	{attribute 'TcIecLibraryType'}
	{attribute 'external_name' := 'F_VN_RotateImageExp2_GUID_B0454A61_6B19_D120_5A5F_16C0F36D78C5'}
	(* Rotate an image by an individual rotation angle in degrees. (expert function) *)
	FUNCTION F_VN_RotateImageExp2 : HRESULT
	VAR_INPUT
		ipSrcImage	:	ITcVnImage;	(* Source image *)
		ipDestImage	:	REFERENCE TO ITcVnImage;	(* Destination image (An appropriate image will be created if required.) *)
		fAngleDeg	:	LREAL;	(* Rotation angle in degree (positive: counter-clockwise, negative: clockwise) *)
		bAdjustDestSize	:	BOOL;	(* If true, ipDestImage size is adjusted so that the whole rotated ipSrcImage is contained. Otherwise, ipDestImage size is set to ipSrcImage size. *)
		eInterpolationType	:	ETcVnInterpolationType;	(* Interpolation method *)
		eBorderInterpolation	:	ETcVnBorderInterpolationMethod;	(* Border interpolation method (ISOLATED not supported) *)
	END_VAR
	VAR_IN_OUT
		aBorderValue	:	TcVnVector4_LREAL;	(* Border value, if CONSTANT is used *)
	END_VAR
	VAR_INPUT
		hrPrev	:	HRESULT;	(* HRESULT indicating the result of previous operations (If SUCCEEDED(hrPrev) equals false, no operation is executed.) *)
	END_VAR

END_FUNCTION

// Functions/Geometric and Coordinate Transformations/F_VN_WarpAffineExp

	{attribute 'TcIecLibraryType'}
	{attribute 'external_name' := 'F_VN_WarpAffineExp_GUID_D07947C7_D823_D73C_7173_E2BD358E148A'}
	(* Apply an affine transformation to an image. (expert function) *)
	FUNCTION F_VN_WarpAffineExp : HRESULT
	VAR_INPUT
		ipSrcImage	:	ITcVnImage;	(* Source image *)
		ipDestImage	:	REFERENCE TO ITcVnImage;	(* Destination image (An appropriate image will be created if required.) *)
	END_VAR
	VAR_IN_OUT
		aTransformationMatrix	:	TcVnMatrix2x3_LREAL;	(* Affine transformation matrix *)
	END_VAR
	VAR_INPUT
		nDestWidth	:	UDINT;	(* Width of the destination image *)
		nDestHeight	:	UDINT;	(* Height of the destination image *)
		eInterpolationType	:	ETcVnInterpolationType;	(* Interpolation method *)
		bWarpInverse	:	BOOL;	(* Handle aTransformationMatrix as the inverse transformation *)
		eBorderInterpolation	:	ETcVnBorderInterpolationMethod;	(* Border interpolation method (ISOLATED not supported) *)
		fBorderValue	:	LREAL;	(* Border value, if CONSTANT is used *)
		hrPrev	:	HRESULT;	(* HRESULT indicating the result of previous operations (If SUCCEEDED(hrPrev) equals false, no operation is executed.) *)
	END_VAR

END_FUNCTION

// Functions/Geometric and Coordinate Transformations/F_VN_WarpAffine_Container

	{attribute 'TcIecLibraryType'}
	{attribute 'external_name' := 'F_VN_WarpAffine_Container_GUID_881050F9_A354_D581_448F_6DB1E8279285'}
	(* Apply an affine transformation to a container of 2D points. *)
	FUNCTION F_VN_WarpAffine_Container : HRESULT
	VAR_INPUT
		ipSrcPoints	:	ITcVnContainer;	(* Source points (ContainerType_Vector_TcVnPoint2_DINT or ContainerType_Vector_TcVnPoint2_REAL or ContainerType_Vector_TcVnPoint2_LREAL) *)
		ipDestPoints	:	REFERENCE TO ITcVnContainer;	(* Returns the transformed points (same type ID as ipSrcPoints; Non-zero interface pointers are reused.) *)
	END_VAR
	VAR_IN_OUT
		aTransformationMatrix	:	TcVnMatrix2x3_LREAL;	(* Affine transformation matrix *)
	END_VAR
	VAR_INPUT
		hrPrev	:	HRESULT;	(* HRESULT indicating the result of previous operations (If SUCCEEDED(hrPrev) equals false, no operation is executed.) *)
	END_VAR

END_FUNCTION

// Functions/Geometric and Coordinate Transformations/F_VN_WarpAffine_Point

	{attribute 'TcIecLibraryType'}
	{attribute 'external_name' := 'F_VN_WarpAffine_Point_GUID_39D72FD9_9F4F_D0F9_78FA_ACBA6F4D42D7'}
	(* Apply an affine transformation to a 2D point. *)
	FUNCTION F_VN_WarpAffine_Point : HRESULT
	VAR_IN_OUT
		aSrcPoint	:	TcVnPoint2_LREAL;	(* Source point *)
		aDestPoint	:	TcVnPoint2_LREAL;	(* Destination point *)
		aTransformationMatrix	:	TcVnMatrix2x3_LREAL;	(* Affine transformation matrix *)
	END_VAR
	VAR_INPUT
		hrPrev	:	HRESULT;	(* HRESULT indicating the result of previous operations (If SUCCEEDED(hrPrev) equals false, no operation is executed.) *)
	END_VAR

END_FUNCTION

// Functions/Geometric and Coordinate Transformations/F_VN_WarpAffine_Rectangle

	{attribute 'TcIecLibraryType'}
	{attribute 'external_name' := 'F_VN_WarpAffine_Rectangle_GUID_69BFAD85_D204_D38A_7FE5_815117E8BF2E'}
	(* Use an affine transform to warp a rectangle. *)
	FUNCTION F_VN_WarpAffine_Rectangle : HRESULT
	VAR_INPUT
		nTopLeftX	:	UDINT;	(* x coordinate of the top left corner *)
		nTopLeftY	:	UDINT;	(* y coordinate of the top left corner *)
		nBottomRightX	:	UDINT;	(* x coordinate of the bottom right corner *)
		nBottomRightY	:	UDINT;	(* y coordinate of the bottom right corner *)
		ipDestPoints	:	REFERENCE TO ITcVnContainer;	(* Returns the 4 transformed points (ContainerType_Vector_TcVnPoint2_REAL) *)
	END_VAR
	VAR_IN_OUT
		aTransformationMatrix	:	TcVnMatrix2x3_LREAL;	(* Affine transformation matrix *)
	END_VAR
	VAR_INPUT
		hrPrev	:	HRESULT;	(* HRESULT indicating the result of previous operations (If SUCCEEDED(hrPrev) equals false, no operation is executed.) *)
	END_VAR

END_FUNCTION

// Functions/Geometric and Coordinate Transformations/F_VN_WarpPerspective

	{attribute 'TcIecLibraryType'}
	{attribute 'external_name' := 'F_VN_WarpPerspective_GUID_CFE51378_A88C_D6F6_6881_5B5CC92D6876'}
	(* Apply a perspective transformation to an image. *)
	FUNCTION F_VN_WarpPerspective : HRESULT
	VAR_INPUT
		ipSrcImage	:	ITcVnImage;	(* Source image *)
		ipDestImage	:	REFERENCE TO ITcVnImage;	(* Destination image (An appropriate image will be created if required.) *)
	END_VAR
	VAR_IN_OUT
		aTransformationMatrix	:	TcVnMatrix3x3_LREAL;	(* Perspective transformation matrix *)
	END_VAR
	VAR_INPUT
		hrPrev	:	HRESULT;	(* HRESULT indicating the result of previous operations (If SUCCEEDED(hrPrev) equals false, no operation is executed.) *)
	END_VAR

END_FUNCTION

// Functions/Geometric and Coordinate Transformations/F_VN_WarpPerspective_Container

	{attribute 'TcIecLibraryType'}
	{attribute 'external_name' := 'F_VN_WarpPerspective_Container_GUID_C43078FC_8F1A_D906_4EBD_0A8B2D834094'}
	(* Apply a perspective transformation to a container of 2D points. *)
	FUNCTION F_VN_WarpPerspective_Container : HRESULT
	VAR_INPUT
		ipSrcPoints	:	ITcVnContainer;	(* Source points (ContainerType_Vector_TcVnPoint2_DINT or ContainerType_Vector_TcVnPoint2_REAL or ContainerType_Vector_TcVnPoint2_LREAL) *)
		ipDestPoints	:	REFERENCE TO ITcVnContainer;	(* Returns the transformed points (same type ID as ipSrcPoints; Non-zero interface pointers are reused.) *)
	END_VAR
	VAR_IN_OUT
		aTransformationMatrix	:	TcVnMatrix3x3_LREAL;	(* Perspective transformation matrix *)
	END_VAR
	VAR_INPUT
		hrPrev	:	HRESULT;	(* HRESULT indicating the result of previous operations (If SUCCEEDED(hrPrev) equals false, no operation is executed.) *)
	END_VAR

END_FUNCTION

// Functions/Geometric and Coordinate Transformations/F_VN_WarpPerspectiveExp

	{attribute 'TcIecLibraryType'}
	{attribute 'external_name' := 'F_VN_WarpPerspectiveExp_GUID_34B331D2_78AA_D3E3_7DC8_94B3A3627598'}
	(* Apply a perspective transformation to an image. (expert function) *)
	FUNCTION F_VN_WarpPerspectiveExp : HRESULT
	VAR_INPUT
		ipSrcImage	:	ITcVnImage;	(* Source image *)
		ipDestImage	:	REFERENCE TO ITcVnImage;	(* Destination image (An appropriate image will be created if required.) *)
	END_VAR
	VAR_IN_OUT
		aTransformationMatrix	:	TcVnMatrix3x3_LREAL;	(* Perspective transformation matrix *)
	END_VAR
	VAR_INPUT
		nDestWidth	:	UDINT;	(* Width of the destination image *)
		nDestHeight	:	UDINT;	(* Height of the destination image *)
		eInterpolationType	:	ETcVnInterpolationType;	(* Interpolation method *)
		bWarpInverse	:	BOOL;	(* Handle aTransformationMatrix as the inverse transformation *)
		eBorderInterpolation	:	ETcVnBorderInterpolationMethod;	(* Border interpolation method (ISOLATED not supported) *)
		fBorderValue	:	LREAL;	(* Border value, if CONSTANT is used *)
		hrPrev	:	HRESULT;	(* HRESULT indicating the result of previous operations (If SUCCEEDED(hrPrev) equals false, no operation is executed.) *)
	END_VAR

END_FUNCTION

// Functions/Geometric and Coordinate Transformations/F_VN_WarpPerspective_Point

	{attribute 'TcIecLibraryType'}
	{attribute 'external_name' := 'F_VN_WarpPerspective_Point_GUID_3F6D0E94_50F7_D140_62FB_6E3EA1ADD95E'}
	(* Apply a perspective transformation to a 2D point. *)
	FUNCTION F_VN_WarpPerspective_Point : HRESULT
	VAR_IN_OUT
		aSrcPoint	:	TcVnPoint2_LREAL;	(* Source point *)
		aDestPoint	:	TcVnPoint2_LREAL;	(* Destination point *)
		aTransformationMatrix	:	TcVnMatrix3x3_LREAL;	(* Perspective transformation matrix *)
	END_VAR
	VAR_INPUT
		hrPrev	:	HRESULT;	(* HRESULT indicating the result of previous operations (If SUCCEEDED(hrPrev) equals false, no operation is executed.) *)
	END_VAR

END_FUNCTION

// Functions/Geometric and Coordinate Transformations/F_VN_WarpPerspective_Rectangle

	{attribute 'TcIecLibraryType'}
	{attribute 'external_name' := 'F_VN_WarpPerspective_Rectangle_GUID_C900301F_B0CF_D57A_7958_23BC0F26B8F7'}
	(* Use a perspective transform to warp a rectangle. *)
	FUNCTION F_VN_WarpPerspective_Rectangle : HRESULT
	VAR_INPUT
		nTopLeftX	:	UDINT;	(* x coordinate of the top left corner *)
		nTopLeftY	:	UDINT;	(* y coordinate of the top left corner *)
		nBottomRightX	:	UDINT;	(* x coordinate of the bottom right corner *)
		nBottomRightY	:	UDINT;	(* y coordinate of the bottom right corner *)
		ipDestPoints	:	REFERENCE TO ITcVnContainer;	(* Returns the 4 transformed points (ContainerType_Vector_TcVnPoint2_REAL) *)
	END_VAR
	VAR_IN_OUT
		aTransformationMatrix	:	TcVnMatrix3x3_LREAL;	(* Perspective transformation matrix *)
	END_VAR
	VAR_INPUT
		hrPrev	:	HRESULT;	(* HRESULT indicating the result of previous operations (If SUCCEEDED(hrPrev) equals false, no operation is executed.) *)
	END_VAR

END_FUNCTION

// Functions/Image Color and Contrast Processing/F_VN_ApplyColorMap

	{attribute 'TcIecLibraryType'}
	{attribute 'external_name' := 'F_VN_ApplyColorMap_GUID_5FC1F56C_5B3C_D465_60AA_C4AA3854379F'}
	(* Apply a color map to a gray-level image. *)
	FUNCTION F_VN_ApplyColorMap : HRESULT
	VAR_INPUT
		ipSrcImage	:	ITcVnImage;	(* Source image (TCVN_ET_USINT or TCVN_ET_UINT, 1 channel) *)
		ipDestImage	:	REFERENCE TO ITcVnImage;	(* Returns the colored image (TCVN_ET_USINT, 3 channel. An appropriate image will be created if required.) *)
		ipColorMap	:	ITcVnContainer;	(* Color map to be applied to ipSrcImage (ContainerType_Vector_TcVnVector3_REAL with 256 or 65536 elements, dependent on ipSrcImage type). Can be either custom or created with F_VN_GenerateColorMap. *)
		hrPrev	:	HRESULT;	(* HRESULT indicating the result of previous operations (If SUCCEEDED(hrPrev) equals false, no operation is executed.) *)
	END_VAR

END_FUNCTION

// Functions/Image Color and Contrast Processing/F_VN_GenerateColorMap

	{attribute 'TcIecLibraryType'}
	{attribute 'external_name' := 'F_VN_GenerateColorMap_GUID_41124A2C_62FC_DD0A_4BF9_B43C26A42D18'}
	(* Generates a pre-defined color map. *)
	FUNCTION F_VN_GenerateColorMap : HRESULT
	VAR_INPUT
		ipColorMap	:	REFERENCE TO ITcVnContainer;	(* Returns the color map (ContainerType_Vector_TcVnVector3_REAL with 256 or 65536 elements) *)
		eColorMap	:	ETcVnColorMap;	(* Selects a color map (similar to GNU Octave/MATLAB types) *)
		eColorMapSize	:	ETcVnColorMapSize;	(* Defines how many elements the generated color map should have *)
		hrPrev	:	HRESULT;	(* HRESULT indicating the result of previous operations (If SUCCEEDED(hrPrev) equals false, no operation is executed.) *)
	END_VAR

END_FUNCTION

// Functions/Image Color and Contrast Processing/F_VN_ApplyLut

	{attribute 'TcIecLibraryType'}
	{attribute 'external_name' := 'F_VN_ApplyLut_GUID_5D73781A_C824_D04E_6F7A_A9EAA2AB4681'}
	(* Apply a lookup table to an image to manipulate its colors. *)
	FUNCTION F_VN_ApplyLut : HRESULT
	VAR_INPUT
		ipSrcImage	:	ITcVnImage;	(* Source image (1-4 channels of 8 or 16 bit types SINT, USINT, INT, UINT) *)
		ipDestImage	:	REFERENCE TO ITcVnImage;	(* Returns the result image (same size, type and channels as ipSrcImage. An appropriate image will be created if required.) *)
		ipLut	:	ITcVnContainer;	(* Lookup table with elements matching ipSrcImage type and either 256 (8 bit images) or 65536 (16 bit images) elements. E.g. ContainerType_Vector_USINT for 1-4 channel USINT image (in this case, the same lookup values are used for each channel) or ContainerType_Vector_TcVnVector3_USINT for a 3 channel USINT image (in this case, each channel uses an individual lookup value).
						 *)
		hrPrev	:	HRESULT;	(* HRESULT indicating the result of previous operations (If SUCCEEDED(hrPrev) equals false, no operation is executed.) *)
	END_VAR

END_FUNCTION

// Functions/Image Color and Contrast Processing/F_VN_Clahe

	{attribute 'TcIecLibraryType'}
	{attribute 'external_name' := 'F_VN_Clahe_GUID_6F92982A_1259_D9E8_5872_BC9EEE361F4F'}
	(* Apply Constrast Limited Adaptive Histogram Equalization. This applies local histogram equalization to individual tiles. *)
	FUNCTION F_VN_Clahe : HRESULT
	VAR_INPUT
		ipSrcImage	:	ITcVnImage;	(* Source image (TCVN_ET_USINT or TCVN_ET_UINT, 1 channel) *)
		ipDestImage	:	REFERENCE TO ITcVnImage;	(* Returns the resulting image (An appropriate image will be created if required.) *)
		hrPrev	:	HRESULT;	(* HRESULT indicating the result of previous operations (If SUCCEEDED(hrPrev) equals false, no operation is executed.) *)
	END_VAR

END_FUNCTION

// Functions/Image Color and Contrast Processing/F_VN_ClaheExp

	{attribute 'TcIecLibraryType'}
	{attribute 'external_name' := 'F_VN_ClaheExp_GUID_D5AEAD88_7973_D98E_640E_FCB90EEA4C61'}
	(* Apply Constrast Limited Adaptive Histogram Equalization. This applies local histogram equalization to individual tiles. (expert function) *)
	FUNCTION F_VN_ClaheExp : HRESULT
	VAR_INPUT
		ipSrcImage	:	ITcVnImage;	(* Source image (TCVN_ET_USINT or TCVN_ET_UINT, 1 channel) *)
		ipDestImage	:	REFERENCE TO ITcVnImage;	(* Returns the resulting image (An appropriate image will be created if required.) *)
		fClipLimit	:	LREAL;	(* Threshold for contrast limit (set to <= 0 to disable clipping) *)
		nTilesX	:	UDINT;	(* Number of tiles in x direction *)
		nTilesY	:	UDINT;	(* Number of tiles in y direction *)
		hrPrev	:	HRESULT;	(* HRESULT indicating the result of previous operations (If SUCCEEDED(hrPrev) equals false, no operation is executed.) *)
	END_VAR

END_FUNCTION

// Functions/Image Color and Contrast Processing/F_VN_ConvertColorSpace

	{attribute 'TcIecLibraryType'}
	{attribute 'external_name' := 'F_VN_ConvertColorSpace_GUID_3928ED09_5286_D091_6CFF_018E8A67A19B'}
	(* Convert image from one color space to another. *)
	FUNCTION F_VN_ConvertColorSpace : HRESULT
	VAR_INPUT
		ipSrcImage	:	ITcVnImage;	(* Source image *)
		ipDestImage	:	REFERENCE TO ITcVnImage;	(* Destination image (An appropriate destination image will be created if required.) *)
		eTransform	:	ETcVnColorSpaceTransform;	(* Transforms to be applied *)
		hrPrev	:	HRESULT;	(* HRESULT indicating the result of previous operations (If SUCCEEDED(hrPrev) equals false, no operation is executed.) *)
	END_VAR

END_FUNCTION

// Functions/Image Color and Contrast Processing/F_VN_GenerateCustomColorMap

	{attribute 'TcIecLibraryType'}
	{attribute 'external_name' := 'F_VN_GenerateCustomColorMap_GUID_25265482_D991_DD20_5A65_7D8187FF081F'}
	(* Generate a custom color map by interpolating between user defined colors (equally distributed, linear for each channel). *)
	FUNCTION F_VN_GenerateCustomColorMap : HRESULT
	VAR_INPUT
		ipColorMap	:	REFERENCE TO ITcVnContainer;	(* Returns the color map (ContainerType_Vector_TcVnVector3_REAL with 256 or 65536 elements) *)
		ipInitialColors	:	ITcVnContainer;	(* User defined colors (ContainerType_Vector_TcVnVector3_REAL, at least 2 elements) *)
		eColorMapSize	:	ETcVnColorMapSize;	(* Defines how many elements the generated color map should have *)
		hrPrev	:	HRESULT;	(* HRESULT indicating the result of previous operations (If SUCCEEDED(hrPrev) equals false, no operation is executed.) *)
	END_VAR

END_FUNCTION

// Functions/Image Color and Contrast Processing/F_VN_Histogram

	{attribute 'TcIecLibraryType'}
	{attribute 'external_name' := 'F_VN_Histogram_GUID_4967AB6E_7C40_DDEE_7ACD_6DC0B6B84EBF'}
	(* Calculate the (multi-channel) histogram of an image. *)
	FUNCTION F_VN_Histogram : HRESULT
	VAR_INPUT
		ipSrcImage	:	ITcVnImage;	(* Source image *)
		ipDestHistogram	:	REFERENCE TO ITcVnContainer;	(* Returns a container with a multi-channel histogram, where every channel is represented as a vector of UDINT (ContainerType_Vector_Vector_UDINT. Non-zero interface pointers are reused.) *)
		hrPrev	:	HRESULT;	(* HRESULT indicating the result of previous operations (If SUCCEEDED(hrPrev) equals false, no operation is executed.) *)
	END_VAR

END_FUNCTION

// Functions/Image Color and Contrast Processing/F_VN_HistogramExp

	{attribute 'TcIecLibraryType'}
	{attribute 'external_name' := 'F_VN_HistogramExp_GUID_C24DCAD7_922F_DA99_5C1A_00E5A61DD4E7'}
	(* Calculate the (multi-channel) histogram of an image. (expert function) *)
	FUNCTION F_VN_HistogramExp : HRESULT
	VAR_INPUT
		ipSrcImage	:	ITcVnImage;	(* Source image *)
		ipDestHistogram	:	REFERENCE TO ITcVnContainer;	(* Returns a container with a multi-channel histogram, where every channel is represented as a vector of UDINT (ContainerType_Vector_Vector_UDINT. Non-zero interface pointers are reused.) *)
	END_VAR
	VAR_IN_OUT
		nBins	:	UDINT;	(* Desired number of bins or 0 to keep the default for the corresponding image format (in) and default number of bins (out) *)
		fLowerBound	:	LREAL;	(* Lower (inclusive) boundary of the 0-th histogram bin (in), or receive the default if fLowerBound AND fUpperBound are set to 0 (out) *)
		fUpperBound	:	LREAL;	(* Upper (exclusive) boundary of the last histogram bin nBins-1 (in), or receive the default if fLowerBound AND fUpperBound are set to 0 (out) *)
	END_VAR
	VAR_INPUT
		ipMask	:	ITcVnImage;	(* Source image mask (TCVN_ET_USINT, 1 channel. Mask is optional, set to 0 if not required.) *)
		hrPrev	:	HRESULT;	(* HRESULT indicating the result of previous operations (If SUCCEEDED(hrPrev) equals false, no operation is executed.) *)
	END_VAR

END_FUNCTION

// Functions/Image Color and Contrast Processing/F_VN_HistogramEqualization

	{attribute 'TcIecLibraryType'}
	{attribute 'external_name' := 'F_VN_HistogramEqualization_GUID_E4A7191D_DEB2_D844_61A1_8D5192620F8A'}
	(* Equalize the histogram of a grayscale or rgb image, which normalizes the brightness and improves the contrast. *)
	FUNCTION F_VN_HistogramEqualization : HRESULT
	VAR_INPUT
		ipSrcImage	:	ITcVnImage;	(* Source image *)
		ipDestImage	:	REFERENCE TO ITcVnImage;	(* Destination image (An appropriate destination image will be created if required.) *)
		hrPrev	:	HRESULT;	(* HRESULT indicating the result of previous operations (If SUCCEEDED(hrPrev) equals false, no operation is executed.) *)
	END_VAR

END_FUNCTION

// Functions/Image Color and Contrast Processing/F_VN_HistogramEqualizationExp

	{attribute 'TcIecLibraryType'}
	{attribute 'external_name' := 'F_VN_HistogramEqualizationExp_GUID_8EB4C057_2479_D74C_4CCA_F2B7F514C2BC'}
	(* Equalize the histogram of a grayscale or color image, which normalizes the brightness and improves the contrast. (expert function) 
	The channel index that should be equalized has to be specified (-1 expects a RGB image, converts it to YCbCr, equalizes the Y channel and converts the image back to RGB).  *)
	FUNCTION F_VN_HistogramEqualizationExp : HRESULT
	VAR_INPUT
		ipSrcImage	:	ITcVnImage;	(* Source image *)
		ipDestImage	:	REFERENCE TO ITcVnImage;	(* Destination image (An appropriate destination image will be created if required.) *)
		nChannelIdx	:	INT;	(* Index of the image channel that should be equalized (-1 expects a RGB image, converts it to YCbCr, equalizes the Y channel and converts the image back to RGB) *)
		hrPrev	:	HRESULT;	(* HRESULT indicating the result of previous operations (If SUCCEEDED(hrPrev) equals false, no operation is executed.) *)
	END_VAR

END_FUNCTION

// Functions/Image Color and Contrast Processing/F_VN_InvertImageColor

	{attribute 'TcIecLibraryType'}
	{attribute 'external_name' := 'F_VN_InvertImageColor_GUID_37BC3565_41C2_D780_6FEB_8C8E78361D97'}
	(* Invert the color of an image.
          For signed integer or negative floating point values, only the signs will be switched.
          If the image contains only positive floating point values, each pixel value is subtracted from the maximum available pixel value (or 1.0, whatever is higher). *)
	FUNCTION F_VN_InvertImageColor : HRESULT
	VAR_INPUT
		ipSrcImage	:	ITcVnImage;	(* Source image *)
		ipDestImage	:	REFERENCE TO ITcVnImage;	(* Destination image (An appropriate image will be created if required.) *)
		hrPrev	:	HRESULT;	(* HRESULT indicating the result of previous operations (If SUCCEEDED(hrPrev) equals false, no operation is executed.) *)
	END_VAR

END_FUNCTION

// Functions/Image Color and Contrast Processing/F_VN_InvertImageColorExp

	{attribute 'TcIecLibraryType'}
	{attribute 'external_name' := 'F_VN_InvertImageColorExp_GUID_D8CA267F_20FA_D72A_5CA4_D061DDB2DC5B'}
	(* Invert the color of an image. (expert function)
          For signed integer or negative floating point values, only the signs will be switched.
          If the image contains only positive floating point values, each pixel value is subtracted from the maximum available pixel value (or 1.0, whatever is higher). *)
	FUNCTION F_VN_InvertImageColorExp : HRESULT
	VAR_INPUT
		ipSrcImage	:	ITcVnImage;	(* Source image *)
		ipDestImage	:	REFERENCE TO ITcVnImage;	(* Destination image (An appropriate image will be created if required.) *)
		fMaxValue	:	LREAL;	(* Maximum pixel value (e.g. if a 16 bit image contains 12 bit values). -1 means the default values are used. *)
		hrPrev	:	HRESULT;	(* HRESULT indicating the result of previous operations (If SUCCEEDED(hrPrev) equals false, no operation is executed.) *)
	END_VAR

END_FUNCTION

// Functions/Image Color and Contrast Processing/F_VN_NormalizeImage

	{attribute 'TcIecLibraryType'}
	{attribute 'external_name' := 'F_VN_NormalizeImage_GUID_01C94C10_A06A_D62A_55A0_B2526D33140F'}
	(* Normalize an image regarding its value range (e.g. stretch pixel values [50..150] to full range [0..255]). *)
	FUNCTION F_VN_NormalizeImage : HRESULT
	VAR_INPUT
		ipSrcImage	:	ITcVnImage;	(* Source image *)
		ipDestImage	:	REFERENCE TO ITcVnImage;	(* Destination image (An appropriate destination image will be created if required.) *)
		hrPrev	:	HRESULT;	(* HRESULT indicating the result of previous operations (If SUCCEEDED(hrPrev) equals false, no operation is executed.) *)
	END_VAR

END_FUNCTION

// Functions/Image Color and Contrast Processing/F_VN_NormalizeImageExp

	{attribute 'TcIecLibraryType'}
	{attribute 'external_name' := 'F_VN_NormalizeImageExp_GUID_F9250BFC_E526_D3A0_70B1_145F0908CE43'}
	(* Normalize an image regarding its value range (e.g. stretch pixel values [50..150] to full range [0..255]) or scale the values regarding a specific normalization (e.g. L2-norm). (expert function) *)
	FUNCTION F_VN_NormalizeImageExp : HRESULT
	VAR_INPUT
		ipSrcImage	:	ITcVnImage;	(* Source image *)
		ipDestImage	:	REFERENCE TO ITcVnImage;	(* Destination image (An appropriate destination image will be created if required.) *)
		fAlpha	:	LREAL;	(* Lower range boundary (in case of normalizing the value range) or value to normalize to (||ipDestImage|| = fAlpha) *)
		fBeta	:	LREAL;	(* Upper range boundary (in case of normalizing the value range) *)
		eNormType	:	ETcVnNormalizationType;	(* Normalization type (only INF, L1, L2 or MINMAX) *)
		eDestType	:	ETcVnElementType;	(* Destination image depth (usually SAME_AS_SOURCE) *)
		ipMask	:	ITcVnImage;	(* Mask to restrict the normalization to specific pixel positions (set 0 to normalize the whole image) *)
		hrPrev	:	HRESULT;	(* HRESULT indicating the result of previous operations (If SUCCEEDED(hrPrev) equals false, no operation is executed.) *)
	END_VAR

END_FUNCTION

// Functions/Image Color and Contrast Processing/F_VN_NormalizeImageForDisplay

	{attribute 'TcIecLibraryType'}
	{attribute 'external_name' := 'F_VN_NormalizeImageForDisplay_GUID_5A39AF93_6FA8_DA77_5213_DA2C848DE791'}
	(* Normalize an image for display, i.e. scale it to the full value range of the underlying data type (-1 to 1 for floating point). *)
	FUNCTION F_VN_NormalizeImageForDisplay : HRESULT
	VAR_INPUT
		ipSrcImage	:	ITcVnImage;	(* Source image *)
		ipDestImage	:	REFERENCE TO ITcVnImage;	(* Destination image (An appropriate destination image will be created if required.) *)
		eSignedNormalization	:	ETcVnSignedNormalization;	(* Option for normalizing signed values *)
		hrPrev	:	HRESULT;	(* HRESULT indicating the result of previous operations (If SUCCEEDED(hrPrev) equals false, no operation is executed.) *)
	END_VAR

END_FUNCTION

// Functions/Image Color and Contrast Processing/F_VN_ReferenceColorSimilarity_ITcVnColorModel

	{attribute 'TcIecLibraryType'}
	{attribute 'external_name' := 'F_VN_ReferenceColorSimilarity_ITcVnColorModel_GUID_2A1F7AC8_C700_D330_6AC5_E4FDC13D131C'}
	(* Computes the similarity to a reference color model for each pixel in the source image. *)
	FUNCTION F_VN_ReferenceColorSimilarity_ITcVnColorModel : HRESULT
	VAR_INPUT
		ipSrcImage	:	ITcVnImage;	(* RGB source image (USINT, 3 channels) *)
		ipDestImage	:	REFERENCE TO ITcVnImage;	(* Returns the similarity to ipColorModel for each pixel in ipSrcImage (USINT, 1 channel. An appropriate destination image will be created if required.) *)
		ipColorModel	:	ITcVnColorModel;	(* Color model *)
		hrPrev	:	HRESULT;	(* HRESULT indicating the result of previous operations (If SUCCEEDED(hrPrev) equals false, no operation is executed.) *)
	END_VAR

END_FUNCTION

// Interfaces/Machine Learning/ITcVnColorModel

	(* Interface to train and classify an image color. *)
	{attribute 'c++_compatible'}
	{attribute 'vtable_order' := 'TrainImageColor;ClassifyImageColor'}
	INTERFACE ITcVnColorModel EXTENDS ITcVnMlModel


(* Train the color of the provided image. *)
	{attribute 'c++_compatible'}
	{attribute 'minimal_input_size' := '4'}
	{attribute 'pack_mode' := '4'}
	METHOD TrainImageColor : HRESULT
	VAR_INPUT
		ipSrcImage : ITcVnImage;
		nDifferentColors : UDINT;
		ipMask : ITcVnImage;
		nSkipPixels : UDINT;
	END_VAR
END_METHOD


(* Compute the similarity of each image pixel to the trained reference color. *)
	{attribute 'c++_compatible'}
	{attribute 'minimal_input_size' := '4'}
	{attribute 'pack_mode' := '4'}
	METHOD ClassifyImageColor : HRESULT
	VAR_INPUT
		ipSrcImage : ITcVnImage;
		pipDestImage : POINTER TO ITcVnImage;
		fVariance : REAL;
		fLuminanceWeight : REAL;
	END_VAR
END_METHOD

END_INTERFACE

// Functions/Image Color and Contrast Processing/F_VN_ReferenceColorSimilarityExp_ITcVnColorModel

	{attribute 'TcIecLibraryType'}
	{attribute 'external_name' := 'F_VN_ReferenceColorSimilarityExp_ITcVnColorModel_GUID_2E034A73_4EF1_D287_407C_3A587C275268'}
	(* Computes the similarity to a reference color model for each pixel in the source image. (expert function) *)
	FUNCTION F_VN_ReferenceColorSimilarityExp_ITcVnColorModel : HRESULT
	VAR_INPUT
		ipSrcImage	:	ITcVnImage;	(* RGB source image (USINT, 3 channels) *)
		ipDestImage	:	REFERENCE TO ITcVnImage;	(* Returns the similarity to ipColorModel for each pixel in ipSrcImage (USINT, 1 channel. An appropriate destination image will be created if required.) *)
		ipColorModel	:	ITcVnColorModel;	(* Color model *)
		fVariance	:	REAL;	(* Allowed color variance (0.1 - 0.3 might be a good start to try) *)
		fLuminanceWeight	:	REAL;	(* Weight the impact of the luminance ([0..1], e.g. set to 0 to be more resistant to unequal illumination, but might be required to differentiate between some colors. Ignored if ipColorModel is of type RGB.) *)
		hrPrev	:	HRESULT;	(* HRESULT indicating the result of previous operations (If SUCCEEDED(hrPrev) equals false, no operation is executed.) *)
	END_VAR

END_FUNCTION

// Functions/Image Color and Contrast Processing/F_VN_ReferenceColorSimilarity_ITcVnMlModel

	{attribute 'TcIecLibraryType'}
	{attribute 'external_name' := 'F_VN_ReferenceColorSimilarity_ITcVnMlModel_GUID_7A720166_859C_DC02_5DA3_02CED4582008'}
	(* Computes the similarity to a reference color model for each pixel in the source image. *)
	FUNCTION F_VN_ReferenceColorSimilarity_ITcVnMlModel : HRESULT
	VAR_INPUT
		ipSrcImage	:	ITcVnImage;	(* RGB source image (USINT, 3 channels) *)
		ipDestImage	:	REFERENCE TO ITcVnImage;	(* Returns the similarity to ipColorModel for each pixel in ipSrcImage (USINT, 1 channel. An appropriate destination image will be created if required.) *)
		ipColorModel	:	ITcVnMlModel;	(* Color model *)
		hrPrev	:	HRESULT;	(* HRESULT indicating the result of previous operations (If SUCCEEDED(hrPrev) equals false, no operation is executed.) *)
	END_VAR

END_FUNCTION

// Functions/Image Color and Contrast Processing/F_VN_ReferenceColorSimilarityExp_ITcVnMlModel

	{attribute 'TcIecLibraryType'}
	{attribute 'external_name' := 'F_VN_ReferenceColorSimilarityExp_ITcVnMlModel_GUID_58AE79C4_8392_D997_6DCA_D06724B6AE4D'}
	(* Computes the similarity to a reference color model for each pixel in the source image. (expert function) *)
	FUNCTION F_VN_ReferenceColorSimilarityExp_ITcVnMlModel : HRESULT
	VAR_INPUT
		ipSrcImage	:	ITcVnImage;	(* RGB source image (USINT, 3 channels) *)
		ipDestImage	:	REFERENCE TO ITcVnImage;	(* Returns the similarity to ipColorModel for each pixel in ipSrcImage (USINT, 1 channel. An appropriate destination image will be created if required.) *)
		ipColorModel	:	ITcVnMlModel;	(* Color model *)
		fVariance	:	REAL;	(* Allowed color variance (0.1 - 0.3 might be a good start to try) *)
		fLuminanceWeight	:	REAL;	(* Weight the impact of the luminance ([0..1], e.g. set to 0 to be more resistant to unequal illumination, but might be required to differentiate between some colors. Ignored if ipColorModel is of type RGB.) *)
		hrPrev	:	HRESULT;	(* HRESULT indicating the result of previous operations (If SUCCEEDED(hrPrev) equals false, no operation is executed.) *)
	END_VAR

END_FUNCTION

// Functions/Image Color and Contrast Processing/F_VN_ReferenceColorSimilarity_TcVnVector3_LREAL

	{attribute 'TcIecLibraryType'}
	{attribute 'external_name' := 'F_VN_ReferenceColorSimilarity_TcVnVector3_LREAL_GUID_FAFF8BBB_F60C_DAC4_5500_10EB08A58633'}
	(* Computes the similarity to a reference color for each pixel in the source image. *)
	FUNCTION F_VN_ReferenceColorSimilarity_TcVnVector3_LREAL : HRESULT
	VAR_INPUT
		ipSrcImage	:	ITcVnImage;	(* RGB source image (USINT, 3 channels) *)
		ipDestImage	:	REFERENCE TO ITcVnImage;	(* Returns the similarity to aRefColor for each pixel in ipSrcImage (USINT, 1 channel. An appropriate destination image will be created if required.) *)
	END_VAR
	VAR_IN_OUT
		aRefColor	:	TcVnVector3_LREAL;	(* Reference color (RGB, [0..255]) *)
	END_VAR
	VAR_INPUT
		hrPrev	:	HRESULT;	(* HRESULT indicating the result of previous operations (If SUCCEEDED(hrPrev) equals false, no operation is executed.) *)
	END_VAR

END_FUNCTION

// Functions/Image Color and Contrast Processing/F_VN_ReferenceColorSimilarityExp_TcVnVector3_LREAL

	{attribute 'TcIecLibraryType'}
	{attribute 'external_name' := 'F_VN_ReferenceColorSimilarityExp_TcVnVector3_LREAL_GUID_D374A0BE_D5EA_D011_61D8_43F8E1C41E27'}
	(* Computes the similarity to a reference color for each pixel in the source image. (expert function) *)
	FUNCTION F_VN_ReferenceColorSimilarityExp_TcVnVector3_LREAL : HRESULT
	VAR_INPUT
		ipSrcImage	:	ITcVnImage;	(* RGB source image (USINT, 3 channels) *)
		ipDestImage	:	REFERENCE TO ITcVnImage;	(* Returns the similarity to aRefColor for each pixel in ipSrcImage (USINT, 1 channel. An appropriate destination image will be created if required.) *)
	END_VAR
	VAR_IN_OUT
		aRefColor	:	TcVnVector3_LREAL;	(* Reference color (RGB, [0..255]) *)
	END_VAR
	VAR_INPUT
		fVariance	:	REAL;	(* Allowed color variance (0.1 - 0.3 might be a good start to try) *)
		fLuminanceWeight	:	REAL;	(* Weight the impact of the luminance ([0..1], e.g. set to 0 to be more resistant to unequal illumination, but might be required to differentiate between some colors) *)
		hrPrev	:	HRESULT;	(* HRESULT indicating the result of previous operations (If SUCCEEDED(hrPrev) equals false, no operation is executed.) *)
	END_VAR

END_FUNCTION

// Functions/Image Color and Contrast Processing/F_VN_TrainImageColor

	{attribute 'TcIecLibraryType'}
	{attribute 'external_name' := 'F_VN_TrainImageColor_GUID_0286D650_F00C_DA59_6156_CB0B6313F883'}
	(* Create a new color model, describing the image color. *)
	FUNCTION F_VN_TrainImageColor : HRESULT
	VAR_INPUT
		ipSrcImage	:	ITcVnImage;	(* Source image (3 channels (RGB) of type USINT) *)
		ipColorModel	:	REFERENCE TO ITcVnColorModel;	(* Returns the color model *)
		nDifferentColors	:	UDINT;	(* Number of different colors to distinguish *)
		hrPrev	:	HRESULT;	(* HRESULT indicating the result of previous operations (If SUCCEEDED(hrPrev) equals false, no operation is executed.) *)
	END_VAR

END_FUNCTION

// Functions/Image Color and Contrast Processing/F_VN_TrainImageColorExp

	{attribute 'TcIecLibraryType'}
	{attribute 'external_name' := 'F_VN_TrainImageColorExp_GUID_615355F9_6BAF_DD2B_4648_974DBAB6D17A'}
	(* Create a new color model, describing the image color. (expert function) *)
	FUNCTION F_VN_TrainImageColorExp : HRESULT
	VAR_INPUT
		ipSrcImage	:	ITcVnImage;	(* Source image (3 channels (RGB) of type USINT) *)
		ipColorModel	:	REFERENCE TO ITcVnColorModel;	(* Returns the color model *)
		nDifferentColors	:	UDINT;	(* Number of different colors to distinguish *)
		eMethod	:	ETcVnColorTrainingMethod;	(* Color training method *)
		ipMask	:	ITcVnImage;	(* Optional image mask (1 channel of type USINT, set to 0 if not required) *)
		nSkipPixels	:	UDINT;	(* Number of pixels to skip between each evaluated color sample (to achieve a better performance). 0 takes every pixel into account and tends to be more accurate. *)
		hrPrev	:	HRESULT;	(* HRESULT indicating the result of previous operations (If SUCCEEDED(hrPrev) equals false, no operation is executed.) *)
	END_VAR

END_FUNCTION

// Functions/Image Color and Contrast Processing/F_VN_TrainImageColorExp2

	{attribute 'TcIecLibraryType'}
	{attribute 'external_name' := 'F_VN_TrainImageColorExp2_GUID_04621000_6349_D589_543F_EA070237B42C'}
	(* Create a new color model, describing the image color. (expert function) *)
	FUNCTION F_VN_TrainImageColorExp2 : HRESULT
	VAR_INPUT
		ipSrcImage	:	ITcVnImage;	(* Source image (3 channels (RGB) of type USINT) *)
		ipColorModel	:	REFERENCE TO ITcVnColorModel;	(* Returns the color model *)
		nDifferentColors	:	UDINT;	(* Maximum number of different colors to distinguish (if LBG is used as a clustering algorithm, the result might have less different colors, depending on nMaxClusterRadius) *)
		eMethod	:	ETcVnColorTrainingMethod;	(* Color training method *)
		ipMask	:	ITcVnImage;	(* Optional image mask (1 channel of type USINT, set to 0 if not required) *)
		nSkipPixels	:	UDINT;	(* Number of pixels to skip between each evaluated color sample (to achieve a better performance). 0 takes every pixel into account and tends to be more accurate. *)
		eClusteringAlgorithm	:	ETcVnClusteringAlgorithm;	(* Clustering algorithm *)
		nMaxClusterRadius	:	DINT;	(* Only used for the LBG clustering algorithm. Maximum allowed radius (> 0) of a single cluster, i.e. clusters with a higher radius will be split into smaller ones, until a global number of nDifferentColors is reached. *)
		bSingleSplitSteps	:	BOOL;	(* Only used for the LBG clustering algorithm. If true, the global optimization is always run after a single cluster has been split. If false, several clusters are split within the same step before applying the global optimization. Applying the global optimization less often is faster, but can lead to less optimal results, especially having 2 nearby clusters that could be represented by 1) *)
		hrPrev	:	HRESULT;	(* HRESULT indicating the result of previous operations (If SUCCEEDED(hrPrev) equals false, no operation is executed.) *)
	END_VAR

END_FUNCTION

// Functions/Image Color and Contrast Processing/F_VN_TrainImageColor_ITcVnMlModel

	{attribute 'TcIecLibraryType'}
	{attribute 'external_name' := 'F_VN_TrainImageColor_ITcVnMlModel_GUID_4985D650_730F_DDD3_537C_883607504684'}
	(* Create a new color model, describing the image color. *)
	FUNCTION F_VN_TrainImageColor_ITcVnMlModel : HRESULT
	VAR_INPUT
		ipSrcImage	:	ITcVnImage;	(* Source image (3 channels (RGB) of type USINT) *)
		ipColorModel	:	REFERENCE TO ITcVnMlModel;	(* Returns the color model *)
		nDifferentColors	:	UDINT;	(* Number of different colors to distinguish *)
		hrPrev	:	HRESULT;	(* HRESULT indicating the result of previous operations (If SUCCEEDED(hrPrev) equals false, no operation is executed.) *)
	END_VAR

END_FUNCTION

// Functions/Image Color and Contrast Processing/F_VN_TrainImageColorExp_ITcVnMlModel

	{attribute 'TcIecLibraryType'}
	{attribute 'external_name' := 'F_VN_TrainImageColorExp_ITcVnMlModel_GUID_EA6BA25E_3C46_DF47_6C6F_22F5A52F9D7A'}
	(* Create a new color model, describing the image color. (expert function) *)
	FUNCTION F_VN_TrainImageColorExp_ITcVnMlModel : HRESULT
	VAR_INPUT
		ipSrcImage	:	ITcVnImage;	(* Source image (3 channels (RGB) of type USINT) *)
		ipColorModel	:	REFERENCE TO ITcVnMlModel;	(* Returns the color model *)
		nDifferentColors	:	UDINT;	(* Number of different colors to distinguish *)
		eMethod	:	ETcVnColorTrainingMethod;	(* Color training method *)
		ipMask	:	ITcVnImage;	(* Optional image mask (1 channel of type USINT, set to 0 if not required) *)
		nSkipPixels	:	UDINT;	(* Number of pixels to skip between each evaluated color sample (to achieve a better performance). 0 takes every pixel into account and tends to be more accurate. *)
		hrPrev	:	HRESULT;	(* HRESULT indicating the result of previous operations (If SUCCEEDED(hrPrev) equals false, no operation is executed.) *)
	END_VAR

END_FUNCTION

// Functions/Image Color and Contrast Processing/F_VN_TrainImageColorExp2_ITcVnMlModel

	{attribute 'TcIecLibraryType'}
	{attribute 'external_name' := 'F_VN_TrainImageColorExp2_ITcVnMlModel_GUID_52511985_90B2_D792_5FB2_139D60A93CCD'}
	(* Create a new color model, describing the image color. (expert function) *)
	FUNCTION F_VN_TrainImageColorExp2_ITcVnMlModel : HRESULT
	VAR_INPUT
		ipSrcImage	:	ITcVnImage;	(* Source image (3 channels (RGB) of type USINT) *)
		ipColorModel	:	REFERENCE TO ITcVnMlModel;	(* Returns the color model *)
		nDifferentColors	:	UDINT;	(* Maximum number of different colors to distinguish (if LBG is used as a clustering algorithm, the result might have less different colors, depending on nMaxClusterRadius) *)
		eMethod	:	ETcVnColorTrainingMethod;	(* Color training method *)
		ipMask	:	ITcVnImage;	(* Optional image mask (1 channel of type USINT, set to 0 if not required) *)
		nSkipPixels	:	UDINT;	(* Number of pixels to skip between each evaluated color sample (to achieve a better performance). 0 takes every pixel into account and tends to be more accurate. *)
		eClusteringAlgorithm	:	ETcVnClusteringAlgorithm;	(* Clustering algorithm *)
		nMaxClusterRadius	:	DINT;	(* Only used for the LBG clustering algorithm. Maximum allowed radius (> 0) of a single cluster, i.e. clusters with a higher radius will be split into smaller ones, until a global number of nDifferentColors is reached. *)
		bSingleSplitSteps	:	BOOL;	(* Only used for the LBG clustering algorithm. If true, the global optimization is always run after a single cluster has been split. If false, several clusters are split within the same step before applying the global optimization. Applying the global optimization less often is faster, but can lead to less optimal results, especially having 2 nearby clusters that could be represented by 1) *)
		hrPrev	:	HRESULT;	(* HRESULT indicating the result of previous operations (If SUCCEEDED(hrPrev) equals false, no operation is executed.) *)
	END_VAR

END_FUNCTION

// Functions/Contour Analysis/F_VN_ApproximatePolygon

	{attribute 'TcIecLibraryType'}
	{attribute 'external_name' := 'F_VN_ApproximatePolygon_GUID_A6759E56_088C_D805_5B13_269319B72382'}
	(* Approximate a contour to a simplified polygon (using the Douglas-Peucker algorithm). *)
	FUNCTION F_VN_ApproximatePolygon : HRESULT
	VAR_INPUT
		ipSrcContour	:	ITcVnContainer;	(* Single contour (ContainerType_Vector_TcVnPoint2_DINT or ContainerType_Vector_TcVnPoint2_REAL; The elements of this container are the points of the contour.) *)
		ipDestContour	:	REFERENCE TO ITcVnContainer;	(* Returns a container which is filled with the approximated polygon points (same type ID as ipSrcContour; Non-zero interface pointers are reused.) *)
		fMaxDist	:	LREAL;	(* Maximum distance between the original contour and its approximation *)
		bClosed	:	BOOL;	(* Specify, if the contour is closed (first and last points connected) or not *)
		hrPrev	:	HRESULT;	(* HRESULT indicating the result of previous operations (If SUCCEEDED(hrPrev) equals false, no operation is executed.) *)
	END_VAR

END_FUNCTION

// Functions/Contour Analysis/F_VN_CheckIfPointIsInsideContour

	{attribute 'TcIecLibraryType'}
	{attribute 'external_name' := 'F_VN_CheckIfPointIsInsideContour_GUID_63709E0D_0FF9_D66E_470E_CA7899E32930'}
	(* Checks if a point is inside a contour (and optionally return the distance to it). *)
	FUNCTION F_VN_CheckIfPointIsInsideContour : HRESULT
	VAR_INPUT
		ipContour	:	ITcVnContainer;	(* Single contour (ContainerType_Vector_TcVnPoint2_DINT or ContainerType_Vector_TcVnPoint2_REAL) *)
	END_VAR
	VAR_IN_OUT
		aPoint	:	TcVnPoint2_REAL;	(* Point position to check *)
		fDist	:	LREAL;	(* Returns the result (> 0: the point is inside the contour; 0: the point is on the contour; < 0: the point is outside the contour) *)
	END_VAR
	VAR_INPUT
		bMeasureDistance	:	BOOL;	(* If true, fDist returns the distance to the nearest contour edge. Otherwise, fDist only returns -1, 0 or +1 (recommended to set to false if the distance is not required, as this is faster). *)
		hrPrev	:	HRESULT;	(* HRESULT indicating the result of previous operations (If SUCCEEDED(hrPrev) equals false, no operation is executed.) *)
	END_VAR

END_FUNCTION

// Functions/Contour Analysis/F_VN_ContourArea

	{attribute 'TcIecLibraryType'}
	{attribute 'external_name' := 'F_VN_ContourArea_GUID_B2BAC4C4_8A74_DF60_6DCB_90E448A196AE'}
	(* Estimate the contour area using Green's formula. *)
	FUNCTION F_VN_ContourArea : HRESULT
	VAR_INPUT
		ipContour	:	ITcVnContainer;	(* Single contour (ContainerType_Vector_TcVnPoint2_DINT or ContainerType_Vector_TcVnPoint2_REAL; The elements of this container are the points of the contour.) *)
	END_VAR
	VAR_IN_OUT
		fArea	:	LREAL;	(* Returns the estimated contour area (The actual contour area may differ depending on the shape of the contour.) *)
	END_VAR
	VAR_INPUT
		hrPrev	:	HRESULT;	(* HRESULT indicating the result of previous operations (If SUCCEEDED(hrPrev) equals false, no operation is executed.) *)
	END_VAR

END_FUNCTION

// Functions/Contour Analysis/F_VN_ContourCenterOfMass

	{attribute 'TcIecLibraryType'}
	{attribute 'external_name' := 'F_VN_ContourCenterOfMass_GUID_0EDE9E95_2E21_DB9F_7A82_6607D561D193'}
	(* Computes the center of mass of a contour. *)
	FUNCTION F_VN_ContourCenterOfMass : HRESULT
	VAR_INPUT
		ipContour	:	ITcVnContainer;	(* Single contour (ContainerType_Vector_TcVnPoint2_DINT or ContainerType_Vector_TcVnPoint2_REAL; The elements of this container are the points of the contour.) *)
	END_VAR
	VAR_IN_OUT
		aCenterOfMass	:	TcVnPoint2_LREAL;	(* Returns the center of mass of the contour *)
	END_VAR
	VAR_INPUT
		hrPrev	:	HRESULT;	(* HRESULT indicating the result of previous operations (If SUCCEEDED(hrPrev) equals false, no operation is executed.) *)
	END_VAR

END_FUNCTION

// Functions/Contour Analysis/F_VN_ContourCircularity

	{attribute 'TcIecLibraryType'}
	{attribute 'external_name' := 'F_VN_ContourCircularity_GUID_F4352892_2BA6_D355_745A_6547990AB3B5'}
	(* Computes the circularity of a contour (1.0: ideal circle, 0.0: straight line). *)
	FUNCTION F_VN_ContourCircularity : HRESULT
	VAR_INPUT
		ipContour	:	ITcVnContainer;	(* Single contour (ContainerType_Vector_TcVnPoint2_DINT or ContainerType_Vector_TcVnPoint2_REAL; The elements of this container are the points of the contour.) *)
	END_VAR
	VAR_IN_OUT
		fCircularity	:	LREAL;	(* Returns the circularity of the contour [0..1] *)
	END_VAR
	VAR_INPUT
		hrPrev	:	HRESULT;	(* HRESULT indicating the result of previous operations (If SUCCEEDED(hrPrev) equals false, no operation is executed.) *)
	END_VAR

END_FUNCTION

// Functions/Contour Analysis/F_VN_ContourConvexity

	{attribute 'TcIecLibraryType'}
	{attribute 'external_name' := 'F_VN_ContourConvexity_GUID_1A5BB2D3_0C2F_D4D6_52FC_6330B90C33FE'}
	(* Computes the convexity of a contour as the ratio between the contour's area and the area of the convex hull (1.0: convex shapes (i.e. rectangle, circle, ..., etc.), 0.0: zero area (i.e. a line or an empty contour)). *)
	FUNCTION F_VN_ContourConvexity : HRESULT
	VAR_INPUT
		ipContour	:	ITcVnContainer;	(* Single contour (ContainerType_Vector_TcVnPoint2_DINT or ContainerType_Vector_TcVnPoint2_REAL; The elements of this container are the points of the contour.) *)
	END_VAR
	VAR_IN_OUT
		fConvexity	:	LREAL;	(* Returns the convexity of the contour [0..1] *)
	END_VAR
	VAR_INPUT
		hrPrev	:	HRESULT;	(* HRESULT indicating the result of previous operations (If SUCCEEDED(hrPrev) equals false, no operation is executed.) *)
	END_VAR

END_FUNCTION

// Functions/Contour Analysis/F_VN_ContourEccentricity

	{attribute 'TcIecLibraryType'}
	{attribute 'external_name' := 'F_VN_ContourEccentricity_GUID_9587B57D_DE28_DA14_5876_CCA34BF0767F'}
	(* Computes the eccentricity of a contour (0.0: circular, 1.0: linear). *)
	FUNCTION F_VN_ContourEccentricity : HRESULT
	VAR_INPUT
		ipContour	:	ITcVnContainer;	(* Single contour (ContainerType_Vector_TcVnPoint2_DINT or ContainerType_Vector_TcVnPoint2_REAL; The elements of this container are the points of the contour.) *)
	END_VAR
	VAR_IN_OUT
		fEccentricity	:	LREAL;	(* Returns the eccentricity of the contour [0..1] *)
	END_VAR
	VAR_INPUT
		hrPrev	:	HRESULT;	(* HRESULT indicating the result of previous operations (If SUCCEEDED(hrPrev) equals false, no operation is executed.) *)
	END_VAR

END_FUNCTION

// Functions/Contour Analysis/F_VN_ContourElongation

	{attribute 'TcIecLibraryType'}
	{attribute 'external_name' := 'F_VN_ContourElongation_GUID_388026DE_0258_DCF7_5E6D_FB28B635C283'}
	(* Computes the elongation factor of a contour. *)
	FUNCTION F_VN_ContourElongation : HRESULT
	VAR_INPUT
		ipContour	:	ITcVnContainer;	(* Single contour (ContainerType_Vector_TcVnPoint2_DINT or ContainerType_Vector_TcVnPoint2_REAL; The elements of this container are the points of the contour.) *)
	END_VAR
	VAR_IN_OUT
		fElongation	:	LREAL;	(* Returns the elongation of the contour *)
	END_VAR
	VAR_INPUT
		hrPrev	:	HRESULT;	(* HRESULT indicating the result of previous operations (If SUCCEEDED(hrPrev) equals false, no operation is executed.) *)
	END_VAR

END_FUNCTION

// Functions/Contour Analysis/F_VN_ContourExtremePoint

	{attribute 'TcIecLibraryType'}
	{attribute 'external_name' := 'F_VN_ContourExtremePoint_GUID_E523A7B1_3850_D553_5547_D7C0475E6454'}
	(* Finds the contour extreme point. *)
	FUNCTION F_VN_ContourExtremePoint : HRESULT
	VAR_INPUT
		ipContour	:	ITcVnContainer;	(* Source container with 2D points (TcVnPoint2_DINT or TcVnPoint2_REAL or TcVnPoint2_LREAL) *)
		eDirection	:	ETcVnExtremePointDirection;	(* Selects the search direction for the extreme point *)
	END_VAR
	VAR_IN_OUT
		aExtremePoint	:	TcVnPoint2_LREAL;	(* Returns the extreme point of the contour, according to eDirection *)
	END_VAR
	VAR_INPUT
		hrPrev	:	HRESULT;	(* HRESULT indicating the result of previous operations (If SUCCEEDED(hrPrev) equals false, no operation is executed.) *)
	END_VAR

END_FUNCTION

// Functions/Contour Analysis/F_VN_ContourInertiaRatio

	{attribute 'TcIecLibraryType'}
	{attribute 'external_name' := 'F_VN_ContourInertiaRatio_GUID_FD98DD7C_34C4_DACB_4FE2_8BB4ACAD9FBC'}
	(* Computes the inertia ratio of a contour which reflects how a contour/shape is elongated (i.e. circle: 1.0, line: 0.0). *)
	FUNCTION F_VN_ContourInertiaRatio : HRESULT
	VAR_INPUT
		ipContour	:	ITcVnContainer;	(* Single contour (ContainerType_Vector_TcVnPoint2_DINT or ContainerType_Vector_TcVnPoint2_REAL; The elements of this container are the points of the contour.) *)
	END_VAR
	VAR_IN_OUT
		fInertiaRatio	:	LREAL;	(* Returns the inertia raio of the contour [0..1] *)
	END_VAR
	VAR_INPUT
		hrPrev	:	HRESULT;	(* HRESULT indicating the result of previous operations (If SUCCEEDED(hrPrev) equals false, no operation is executed.) *)
	END_VAR

END_FUNCTION

// Functions/Contour Analysis/F_VN_ContourMoments

	{attribute 'TcIecLibraryType'}
	{attribute 'external_name' := 'F_VN_ContourMoments_GUID_909C5166_02C5_D2B0_5963_CBC384FA8873'}
	(* Computes the spatial moments, the central moments, and the central normalized moments of a contour up to the third order. *)
	FUNCTION F_VN_ContourMoments : HRESULT
	VAR_INPUT
		ipContour	:	ITcVnContainer;	(* Single contour (ContainerType_Vector_TcVnPoint2_DINT or ContainerType_Vector_TcVnPoint2_REAL; The elements of this container are the points of the contour.) *)
	END_VAR
	VAR_IN_OUT
		stMoments	:	TcVnMoments;	(* Returns a struct containing the moments *)
	END_VAR
	VAR_INPUT
		hrPrev	:	HRESULT;	(* HRESULT indicating the result of previous operations (If SUCCEEDED(hrPrev) equals false, no operation is executed.) *)
	END_VAR

END_FUNCTION

// Functions/Contour Analysis/F_VN_ContourOrientation

	{attribute 'TcIecLibraryType'}
	{attribute 'external_name' := 'F_VN_ContourOrientation_GUID_E49B3606_6808_D0D0_6E4C_8E27231AAC03'}
	(* Calculate the orientation of a contour or a set of points. *)
	FUNCTION F_VN_ContourOrientation : HRESULT
	VAR_INPUT
		ipContour	:	ITcVnContainer;	(* Source point set (ContainerType_Vector_TcVnPoint2_DINT, ContainerType_Vector_TcVnPoint2_REAL, or ContainerType_Vector_TcVnPoint2_LREAL. The elements of this container are the individual points.) *)
	END_VAR
	VAR_IN_OUT
		stOrientation	:	TcVnRotatedRectangle;	(* Resulting rotated rectangle, containig center of mass, lenghts of axes, and rotation angle of the contour in clockwise direction. *)
	END_VAR
	VAR_INPUT
		hrPrev	:	HRESULT;	(* HRESULT indicating the result of previous operations (If SUCCEEDED(hrPrev) equals false, no operation is executed.) *)
	END_VAR

END_FUNCTION

// Functions/Contour Analysis/F_VN_ContourOrientationExp

	{attribute 'TcIecLibraryType'}
	{attribute 'external_name' := 'F_VN_ContourOrientationExp_GUID_30BB8957_A8B7_D240_40D3_7007CEAB99BB'}
	(* Calculate the orientation of a contour or a set of points. (expert function) *)
	FUNCTION F_VN_ContourOrientationExp : HRESULT
	VAR_INPUT
		ipContour	:	ITcVnContainer;	(* Source point set (ContainerType_Vector_TcVnPoint2_DINT, ContainerType_Vector_TcVnPoint2_REAL, or ContainerType_Vector_TcVnPoint2_LREAL. The elements of this container are the individual points.) *)
	END_VAR
	VAR_IN_OUT
		stOrientation	:	TcVnRotatedRectangle;	(* Resulting rotated rectangle, containig center of mass, lenghts of axes, and rotation angle of the contour in clockwise direction. *)
	END_VAR
	VAR_INPUT
		eMethod	:	ETcVnOrientationMethod;	(* Method for calculating the orientation.  *)
		hrPrev	:	HRESULT;	(* HRESULT indicating the result of previous operations (If SUCCEEDED(hrPrev) equals false, no operation is executed.) *)
	END_VAR

END_FUNCTION

// Functions/Contour Analysis/F_VN_ContourPerimeter

	{attribute 'TcIecLibraryType'}
	{attribute 'external_name' := 'F_VN_ContourPerimeter_GUID_A0075933_8A46_D67D_5D84_0ABAEF182F14'}
	(* Computes the perimeter of a contour (curve length if the contour is not closed). *)
	FUNCTION F_VN_ContourPerimeter : HRESULT
	VAR_INPUT
		ipContour	:	ITcVnContainer;	(* Single contour (ContainerType_Vector_TcVnPoint2_DINT or ContainerType_Vector_TcVnPoint2_REAL; The elements of this container are the points of the contour.) *)
	END_VAR
	VAR_IN_OUT
		fPerimeter	:	LREAL;	(* Returns the perimeter of the contour *)
	END_VAR
	VAR_INPUT
		bClosed	:	BOOL;	(* Specifys, if the contour is closed (first and last points connected) or not *)
		hrPrev	:	HRESULT;	(* HRESULT indicating the result of previous operations (If SUCCEEDED(hrPrev) equals false, no operation is executed.) *)
	END_VAR

END_FUNCTION

// Functions/Contour Analysis/F_VN_ContourRoundness

	{attribute 'TcIecLibraryType'}
	{attribute 'external_name' := 'F_VN_ContourRoundness_GUID_637468D7_1811_DFC5_43AD_833D133AA763'}
	(* Computes the roundness of a contour (perimeter^2 / area). *)
	FUNCTION F_VN_ContourRoundness : HRESULT
	VAR_INPUT
		ipContour	:	ITcVnContainer;	(* Single contour (ContainerType_Vector_TcVnPoint2_DINT or ContainerType_Vector_TcVnPoint2_REAL; The elements of this container are the points of the contour.) *)
	END_VAR
	VAR_IN_OUT
		fRoundness	:	LREAL;	(* Returns the roundness of the contour *)
	END_VAR
	VAR_INPUT
		hrPrev	:	HRESULT;	(* HRESULT indicating the result of previous operations (If SUCCEEDED(hrPrev) equals false, no operation is executed.) *)
	END_VAR

END_FUNCTION

// Functions/Contour Analysis/F_VN_ConvexHullPoints

	{attribute 'TcIecLibraryType'}
	{attribute 'external_name' := 'F_VN_ConvexHullPoints_GUID_39D37EFE_AF46_DF3B_5911_075036B2AE77'}
	(* Determines the convex hull of a point set. *)
	FUNCTION F_VN_ConvexHullPoints : HRESULT
	VAR_INPUT
		ipPointSet	:	ITcVnContainer;	(* Source point set (ContainerType_Vector_TcVnPoint2_DINT or ContainerType_Vector_TcVnPoint2_REAL; The elements of this container are the individual points.) *)
		ipConvexHull	:	REFERENCE TO ITcVnContainer;	(* Returns a container which is filled with the sorted convex hull points (same type ID as ipPointSet; Non-zero interface pointers are reused.) *)
		hrPrev	:	HRESULT;	(* HRESULT indicating the result of previous operations (If SUCCEEDED(hrPrev) equals false, no operation is executed.) *)
	END_VAR

END_FUNCTION

// Functions/Contour Analysis/F_VN_ConvexHullPointsExp

	{attribute 'TcIecLibraryType'}
	{attribute 'external_name' := 'F_VN_ConvexHullPointsExp_GUID_7463719C_F330_D86E_668B_825EE0E4679E'}
	(* Determines the convex hull of a point set. (expert function) *)
	FUNCTION F_VN_ConvexHullPointsExp : HRESULT
	VAR_INPUT
		ipPointSet	:	ITcVnContainer;	(* Source point set (ContainerType_Vector_TcVnPoint2_DINT or ContainerType_Vector_TcVnPoint2_REAL; The elements of this container are the individual points.) *)
		ipConvexHull	:	REFERENCE TO ITcVnContainer;	(* Returns a container which is filled with the sorted convex hull points (same type ID as ipPointSet; Non-zero interface pointers are reused.) *)
		bClockwise	:	BOOL;	(* Selects the sorting direction of the hull points, assuming cartesian coordinates. *)
		hrPrev	:	HRESULT;	(* HRESULT indicating the result of previous operations (If SUCCEEDED(hrPrev) equals false, no operation is executed.) *)
	END_VAR

END_FUNCTION

// Functions/Contour Analysis/F_VN_ConvexityDefects

	{attribute 'TcIecLibraryType'}
	{attribute 'external_name' := 'F_VN_ConvexityDefects_GUID_BEC1372C_18C6_D92E_52DF_CD82B0D46DFD'}
	(* Finds the convexity defects of a point set. *)
	FUNCTION F_VN_ConvexityDefects : HRESULT
	VAR_INPUT
		ipContour	:	ITcVnContainer;	(* Source contour (ContainerType_Vector_TcVnPoint2_DINT; The elements of this container are the individual points.) *)
		ipConvexityDefects	:	REFERENCE TO ITcVnContainer;	(* Returns a container which is filled with the convexity defects (ContainerType_Vector_TcVnVector4_DINT with [startIndex, endIndex, furthestPointIndex, fixedPointDistance (8 fraction bits, i.e. divide by 256 to get the distance in pixels)]; Non-zero interface pointers are reused.) *)
		hrPrev	:	HRESULT;	(* HRESULT indicating the result of previous operations (If SUCCEEDED(hrPrev) equals false, no operation is executed.) *)
	END_VAR

END_FUNCTION

// Functions/Contour Analysis/F_VN_CustomElementWiseContainerOperation_ITcVnContainer

	{attribute 'TcIecLibraryType'}
	{attribute 'external_name' := 'F_VN_CustomElementWiseContainerOperation_ITcVnContainer_GUID_E10A4324_256D_D75D_6CE1_D8055216E65E'}
	(* Performs a custom, element wise operation on a set of up to 3 containers. *)
	FUNCTION F_VN_CustomElementWiseContainerOperation_ITcVnContainer : HRESULT
	VAR_INPUT
		ipContainer1	:	ITcVnContainer;	(* Container 1 *)
		ipContainer2	:	ITcVnContainer;	(* Container 2 *)
		ipContainer3	:	ITcVnContainer;	(* Container 3 *)
		ipOperationFB	:	ITcVnCustomContainerOperation_ITcVnContainer;	(* Custom operation on the container elements *)
		hrPrev	:	HRESULT;	(* HRESULT indicating the result of previous operations (If SUCCEEDED(hrPrev) equals false, no operation is executed.) *)
	END_VAR

END_FUNCTION

// Interfaces/Containers/Function Blocks/ITcVnCustomContainerOperation_ITcVnContainer

	(* Offers an interface for custom, elementwise container operations (for containers of containers) with up to 3 different containers. *)
	{attribute 'c++_compatible'}
	INTERFACE ITcVnCustomContainerOperation_ITcVnContainer


(* Executes the custom operation on the container elements. *)
	{attribute 'c++_compatible'}
	{attribute 'minimal_input_size' := '4'}
	{attribute 'pack_mode' := '4'}
	METHOD Execute : HRESULT
	VAR_INPUT
		ipElement1 : ITcVnContainer;
		ipElement2 : ITcVnContainer;
		ipElement3 : ITcVnContainer;
	END_VAR
END_METHOD

END_INTERFACE

// Functions/Contour Analysis/F_VN_CustomElementWiseContainerOperation_ITcVnForwardIterator

	{attribute 'TcIecLibraryType'}
	{attribute 'external_name' := 'F_VN_CustomElementWiseContainerOperation_ITcVnForwardIterator_GUID_C9A075D3_4499_D759_7B14_F843AE4052E7'}
	(* Performs a custom, element wise operation on a set of up to 3 containers. *)
	FUNCTION F_VN_CustomElementWiseContainerOperation_ITcVnForwardIterator : HRESULT
	VAR_INPUT
		ipContainer1	:	ITcVnContainer;	(* Container 1 *)
		ipContainer2	:	ITcVnContainer;	(* Container 2 *)
		ipContainer3	:	ITcVnContainer;	(* Container 3 *)
		ipOperationFB	:	ITcVnCustomContainerOperation_ITcVnForwardIterator;	(* Custom operation on the elements *)
		hrPrev	:	HRESULT;	(* HRESULT indicating the result of previous operations (If SUCCEEDED(hrPrev) equals false, no operation is executed.) *)
	END_VAR

END_FUNCTION

// Interfaces/Containers/Function Blocks/ITcVnCustomContainerOperation_ITcVnForwardIterator

	(* Offers an interface for custom, elementwise container operations with up to 3 different containers. *)
	{attribute 'c++_compatible'}
	INTERFACE ITcVnCustomContainerOperation_ITcVnForwardIterator


(* Executes the custom operation on the container elements. *)
	{attribute 'c++_compatible'}
	{attribute 'minimal_input_size' := '4'}
	{attribute 'pack_mode' := '4'}
	METHOD Execute : HRESULT
	VAR_INPUT
		ipElement1 : ITcVnForwardIterator;
		ipElement2 : ITcVnForwardIterator;
		ipElement3 : ITcVnForwardIterator;
	END_VAR
END_METHOD

END_INTERFACE

// Functions/Contour Analysis/F_VN_EnclosingCircle

	{attribute 'TcIecLibraryType'}
	{attribute 'external_name' := 'F_VN_EnclosingCircle_GUID_461C7A6E_04DA_DECE_6D16_CA70F1AC8532'}
	(* Searchs for a minimum area circle enclosing a set of points. *)
	FUNCTION F_VN_EnclosingCircle : HRESULT
	VAR_INPUT
		ipPointSet	:	ITcVnContainer;	(* Source point set (ContainerType_Vector_TcVnPoint2_DINT or ContainerType_Vector_TcVnPoint2_REAL; The elements of this container are the individual points.) *)
	END_VAR
	VAR_IN_OUT
		aCenter	:	TcVnPoint2_REAL;	(* Returns the center of the circle *)
		fRadius	:	REAL;	(* Returns the radius of the circle *)
	END_VAR
	VAR_INPUT
		hrPrev	:	HRESULT;	(* HRESULT indicating the result of previous operations (If SUCCEEDED(hrPrev) equals false, no operation is executed.) *)
	END_VAR

END_FUNCTION

// Functions/Contour Analysis/F_VN_EnclosingRectangle

	{attribute 'TcIecLibraryType'}
	{attribute 'external_name' := 'F_VN_EnclosingRectangle_GUID_304B1A1D_A3CD_DAA1_7550_EB825B6C82B2'}
	(* Searches for a minimum area rectangle enclosing a set of points. *)
	FUNCTION F_VN_EnclosingRectangle : HRESULT
	VAR_INPUT
		ipPointSet	:	ITcVnContainer;	(* Source point set (ContainerType_Vector_TcVnPoint2_DINT or ContainerType_Vector_TcVnPoint2_REAL; The elements of this container are the individual points.) *)
	END_VAR
	VAR_IN_OUT
		stRectangle	:	TcVnRotatedRectangle;	(* Returns the determined rectangle *)
	END_VAR
	VAR_INPUT
		hrPrev	:	HRESULT;	(* HRESULT indicating the result of previous operations (If SUCCEEDED(hrPrev) equals false, no operation is executed.) *)
	END_VAR

END_FUNCTION

// Functions/Contour Analysis/F_VN_EnclosingTriangle

	{attribute 'TcIecLibraryType'}
	{attribute 'external_name' := 'F_VN_EnclosingTriangle_GUID_FDB7B043_7F27_D4DE_50FF_890BA9C41B48'}
	(* Searches for a minimum area triangle enclosing a set of points. *)
	FUNCTION F_VN_EnclosingTriangle : HRESULT
	VAR_INPUT
		ipPointSet	:	ITcVnContainer;	(* Source point set (ContainerType_Vector_TcVnPoint2_DINT or ContainerType_Vector_TcVnPoint2_REAL; The elements of this container are the individual points.) *)
	END_VAR
	VAR_IN_OUT
		aTriangleVertices	:	TcVnArray3_Point2_REAL;	(* Returns the 3 triangle vertices *)
	END_VAR
	VAR_INPUT
		hrPrev	:	HRESULT;	(* HRESULT indicating the result of previous operations (If SUCCEEDED(hrPrev) equals false, no operation is executed.) *)
	END_VAR
	VAR_OUTPUT
		fArea	:	LREAL;	(* Returns the triangle area *)
	END_VAR

END_FUNCTION

// Functions/Contour Analysis/F_VN_FitEllipse

	{attribute 'TcIecLibraryType'}
	{attribute 'external_name' := 'F_VN_FitEllipse_GUID_FB03990C_F20D_DE7C_6C62_608DC759EB06'}
	(* Fit an ellipse in a point set. *)
	FUNCTION F_VN_FitEllipse : HRESULT
	VAR_INPUT
		ipPointSet	:	ITcVnContainer;	(* Source point set (ContainerType_Vector_TcVnPoint2_DINT or ContainerType_Vector_TcVnPoint2_REAL; At least 5 reasonable points are required! The elements of this container are the individual points.) *)
	END_VAR
	VAR_IN_OUT
		stEllipse	:	TcVnRotatedRectangle;	(* Resulting ellipse, described by a rotated rectangle. *)
	END_VAR
	VAR_INPUT
		hrPrev	:	HRESULT;	(* HRESULT indicating the result of previous operations (If SUCCEEDED(hrPrev) equals false, no operation is executed.) *)
	END_VAR

END_FUNCTION

// Functions/Contour Analysis/F_VN_FitLine

	{attribute 'TcIecLibraryType'}
	{attribute 'external_name' := 'F_VN_FitLine_GUID_DB152F5D_C12B_D54B_4984_3BD9757F4AA3'}
	(* Fit a line into a point set. *)
	FUNCTION F_VN_FitLine : HRESULT
	VAR_INPUT
		ipPointSet	:	ITcVnContainer;	(* Source point set (ContainerType_Vector_TcVnPoint2_DINT or ContainerType_Vector_TcVnPoint2_REAL; The elements of this container are the individual points.) *)
	END_VAR
	VAR_IN_OUT
		aFitLine	:	TcVnVector4_LREAL;	(* Resulting line. The first and second element describe the x and y component of a vector collinear to the line. The third and fourth element describe the x and y component of a point on the line. *)
	END_VAR
	VAR_INPUT
		hrPrev	:	HRESULT;	(* HRESULT indicating the result of previous operations (If SUCCEEDED(hrPrev) equals false, no operation is executed.) *)
	END_VAR

END_FUNCTION

// Functions/Contour Analysis/F_VN_FitLineExp

	{attribute 'TcIecLibraryType'}
	{attribute 'external_name' := 'F_VN_FitLineExp_GUID_13DE2AA7_E400_DEEC_7138_F5CDA092FCD7'}
	(* Fit a line into a point set. (expert function) *)
	FUNCTION F_VN_FitLineExp : HRESULT
	VAR_INPUT
		ipPointSet	:	ITcVnContainer;	(* Source point set (ContainerType_Vector_TcVnPoint2_DINT or ContainerType_Vector_TcVnPoint2_REAL; The elements of this container are the individual points.) *)
	END_VAR
	VAR_IN_OUT
		aFitLine	:	TcVnVector4_LREAL;	(* Resulting line. The first and second element describe the x and y component of a vector collinear to the line. The third and fourth element describe the x and y component of a point on the line. *)
	END_VAR
	VAR_INPUT
		eDistanceType	:	ETcVnDistanceType;	(* Distance computation method (supported: L1, L2, L12, FAIR, WELSCH, HUBER) *)
		fParam	:	LREAL;	(* Numerical parameter (c) for some eDistanceType (should be >= 0). If 0, an optimal value is chosen internally. *)
		fEpsRadius	:	LREAL;	(* Accuracy of the radius (distance of the line from the coordinate origin, should be > 0). A smaller value means higher accuracy. *)
		fEpsAngle	:	LREAL;	(* Accuracy of the angle (should be > 0). A smaller value means higher accuracy. *)
		hrPrev	:	HRESULT;	(* HRESULT indicating the result of previous operations (If SUCCEEDED(hrPrev) equals false, no operation is executed.) *)
	END_VAR

END_FUNCTION

// Functions/Contour Analysis/F_VN_FourierDescriptors

	{attribute 'TcIecLibraryType'}
	{attribute 'external_name' := 'F_VN_FourierDescriptors_GUID_4264AD18_43DA_D302_5AB5_01A5356BDD2B'}
	(* Computes the fourier descriptors for a closed contour. *)
	FUNCTION F_VN_FourierDescriptors : HRESULT
	VAR_INPUT
		ipContour	:	ITcVnContainer;	(* Closed contour (ContainerType_Vector_TcVnPoint2_DINT or ContainerType_Vector_TcVnPoint2_REAL or ContainerType_Vector_TcVnPoint2_LREAL. Providing the full contour is strongly recommended, i.e. use TCVN_CAM_NONE for contour detection algorithms.) *)
		ipDescriptors	:	REFERENCE TO ITcVnContainer;	(* Returns the fourier descriptors for ipContour (Re0, Im0, Re1, Im1, ...; ContainerType_Vector_LREAL if ipContour is of type ContainerType_Vector_TcVnPoint2_LREAL, else ContainerType_Vector_REAL.) *)
		nDescriptors	:	DINT;	(* Specifies how many descriptors should be returned (set to -1 to return all computed descriptors, i.e. at least as many as the number of contour points) *)
		hrPrev	:	HRESULT;	(* HRESULT indicating the result of previous operations (If SUCCEEDED(hrPrev) equals false, no operation is executed.) *)
	END_VAR

END_FUNCTION

// Functions/Contour Analysis/F_VN_MatchContours

	{attribute 'TcIecLibraryType'}
	{attribute 'external_name' := 'F_VN_MatchContours_GUID_ADEFFFA4_843C_D220_5FCD_C2AF67E4288E'}
	(* Compare contours using the Hu moment invariants. In case of multiple contours in each container, the best matches are found and the average dissimilarity over all matched contours is returned. *)
	FUNCTION F_VN_MatchContours : HRESULT
	VAR_INPUT
		ipContour1	:	ITcVnContainer;	(* First contour (ContainerType_Vector_TcVnPoint2_DINT or ContainerType_Vector_TcVnPoint2_REAL; The elements of this container are the points of the contour) or collection of multiple contours (ContainerType_Vector_Vector_TcVnPoint2_DINT) *)
		ipContour2	:	ITcVnContainer;	(* Second contour (same type as ipContour1) *)
		eComparisonMethod	:	ETcVnContoursMatchComparisonMethod;	(* Method used for comparing the Hu moment invariants of the contours *)
	END_VAR
	VAR_IN_OUT
		fDissimilarity	:	LREAL;	(* Returns the dissimilarity of the contours depending on the chosen comparison method *)
	END_VAR
	VAR_INPUT
		hrPrev	:	HRESULT;	(* HRESULT indicating the result of previous operations (If SUCCEEDED(hrPrev) equals false, no operation is executed.) *)
	END_VAR

END_FUNCTION

// Functions/Contour Analysis/F_VN_MatchContoursExp

	{attribute 'TcIecLibraryType'}
	{attribute 'external_name' := 'F_VN_MatchContoursExp_GUID_DC94C6D0_8BB0_DA38_592C_A63A4568E0E9'}
	(* Compare contours using the Hu moment invariants (and optionally further aspects). In case of multiple contours in each container, the best matches are found and the average dissimilarity over all matched contours is returned. (expert function) *)
	FUNCTION F_VN_MatchContoursExp : HRESULT
	VAR_INPUT
		ipContour1	:	ITcVnContainer;	(* First contour (ContainerType_Vector_TcVnPoint2_DINT or ContainerType_Vector_TcVnPoint2_REAL; The elements of this container are the points of the contour) or collection of multiple contours (ContainerType_Vector_Vector_TcVnPoint2_DINT) *)
		ipContour2	:	ITcVnContainer;	(* Second contour (same type as ipContour1) *)
		eComparisonMethod	:	ETcVnContoursMatchComparisonMethod;	(* Method used for comparing the Hu moment invariants of the contours *)
	END_VAR
	VAR_IN_OUT
		fDissimilarity	:	LREAL;	(* Returns the dissimilarity of the contours depending on the chosen comparison method *)
	END_VAR
	VAR_INPUT
		fAreaFactor	:	LREAL;	(* If > 0, the relative area difference between contours is scaled by this factor and added to the computed dissimilarity *)
		fAbsPositionFactor	:	LREAL;	(* If > 0, the absolute position difference between contours (i.e. the coordinates of the geometric contour centers) is scaled by this factor and added to the computed dissimilarity *)
		fRelPositionFactor	:	LREAL;	(* If > 0, the relative position difference between contours is scaled by this factor and added to the computed dissimilarity (only used if matching multiple contours) *)
		fNumDiffFactor	:	LREAL;	(* If > 0, the difference between the number of contours in both containers is scaled by this factor and added to the computed dissimilarity (only used if matching multiple contours) *)
		hrPrev	:	HRESULT;	(* HRESULT indicating the result of previous operations (If SUCCEEDED(hrPrev) equals false, no operation is executed.) *)
	END_VAR

END_FUNCTION

// Functions/Contour Analysis/F_VN_MatchContours1vsN

	{attribute 'TcIecLibraryType'}
	{attribute 'external_name' := 'F_VN_MatchContours1vsN_GUID_14D953BB_F4B3_D80A_6815_21EA7C8E49AB'}
	(* Compare a reference contour with multiple other contours using the Hu moment invariants. Returns a sorted list of best matches. *)
	FUNCTION F_VN_MatchContours1vsN : HRESULT
	VAR_INPUT
		ipRefContour	:	ITcVnContainer;	(* Reference contour (ContainerType_Vector_TcVnPoint2_DINT or ContainerType_Vector_TcVnPoint2_REAL; The elements of this container are the points of the contour) *)
		ipContours	:	ITcVnContainer;	(* Collection of multiple contours (CTcVnContainer_Vector_Vector_TcVnPoint2_DINT) *)
		ipMatchIndexes	:	REFERENCE TO ITcVnContainer;	(* Returns the indexes of the best matches (CTcVnContainer_Vector_ULINT; sorted, first element is best match, i.e. has lowest dissimilarity) *)
		ipDissimilarities	:	REFERENCE TO ITcVnContainer;	(* Returns the computed dissimilarities of the best matches (CTcVnContainer_Vector_LREAL; Optional, set to 0 if not required; sorted corresponding to ipMatchIndexes) *)
		fDissimilarityThreshold	:	LREAL;	(* Neglect irrelevant matches, i.e. dissimilarity > fDissimilarityThreshold *)
		eComparisonMethod	:	ETcVnContoursMatchComparisonMethod;	(* Method used for comparing the Hu moment invariants of the contours *)
		hrPrev	:	HRESULT;	(* HRESULT indicating the result of previous operations (If SUCCEEDED(hrPrev) equals false, no operation is executed.) *)
	END_VAR

END_FUNCTION

// Functions/Contour Analysis/F_VN_MatchContours1vsNExp

	{attribute 'TcIecLibraryType'}
	{attribute 'external_name' := 'F_VN_MatchContours1vsNExp_GUID_598D2F5E_7AEB_D303_5812_05F0E90142E6'}
	(* Compare a reference contour with multiple other contours using the Hu moment invariants (and optionally further aspects). Returns a sorted list of best matches. (expert function) *)
	FUNCTION F_VN_MatchContours1vsNExp : HRESULT
	VAR_INPUT
		ipRefContour	:	ITcVnContainer;	(* Reference contour (ContainerType_Vector_TcVnPoint2_DINT or ContainerType_Vector_TcVnPoint2_REAL; The elements of this container are the points of the contour) *)
		ipContours	:	ITcVnContainer;	(* Collection of multiple contours (CTcVnContainer_Vector_Vector_TcVnPoint2_DINT) *)
		ipMatchIndexes	:	REFERENCE TO ITcVnContainer;	(* Returns the indexes of the best matches (CTcVnContainer_Vector_ULINT; sorted, first element is best match, i.e. has lowest dissimilarity) *)
		ipDissimilarities	:	REFERENCE TO ITcVnContainer;	(* Returns the computed dissimilarities of the best matches (CTcVnContainer_Vector_LREAL; Optional, set to 0 if not required; sorted corresponding to ipMatchIndexes) *)
		fDissimilarityThreshold	:	LREAL;	(* Neglect irrelevant matches, i.e. dissimilarity > fDissimilarityThreshold *)
		eComparisonMethod	:	ETcVnContoursMatchComparisonMethod;	(* Method used for comparing the Hu moment invariants of the contours *)
		fAreaFactor	:	LREAL;	(* If > 0, the relative area difference between contours is scaled by this factor and added to the computed dissimilarity *)
		fAbsPositionFactor	:	LREAL;	(* If > 0, the absolute position difference between contours (i.e. the coordinates of the geometric contour centers) is scaled by this factor and added to the computed dissimilarity *)
		hrPrev	:	HRESULT;	(* HRESULT indicating the result of previous operations (If SUCCEEDED(hrPrev) equals false, no operation is executed.) *)
	END_VAR

END_FUNCTION

// Functions/Contour Analysis/F_VN_UprightBoundingRectangle

	{attribute 'TcIecLibraryType'}
	{attribute 'external_name' := 'F_VN_UprightBoundingRectangle_GUID_1A75DA06_689D_D5B6_459A_F1682FC8D247'}
	(* Determines the upright bounding rectangle of a set of points. *)
	FUNCTION F_VN_UprightBoundingRectangle : HRESULT
	VAR_INPUT
		ipPointSet	:	ITcVnContainer;	(* Source point set (ContainerType_Vector_TcVnPoint2_DINT or ContainerType_Vector_TcVnPoint2_REAL; The elements of this container are the individual points.) *)
	END_VAR
	VAR_IN_OUT
		stRectangle	:	TcVnRectangle_UDINT;	(* Returns the determined rectangle *)
	END_VAR
	VAR_INPUT
		hrPrev	:	HRESULT;	(* HRESULT indicating the result of previous operations (If SUCCEEDED(hrPrev) equals false, no operation is executed.) *)
	END_VAR

END_FUNCTION

// Functions/Image Filtering/F_VN_BilateralFilter

	{attribute 'TcIecLibraryType'}
	{attribute 'external_name' := 'F_VN_BilateralFilter_GUID_21B5D26A_DD92_D49B_49C0_1C2A6673355D'}
	(* Apply a Bilateral filter to smooth the image but preserve edges. *)
	FUNCTION F_VN_BilateralFilter : HRESULT
	VAR_INPUT
		ipSrcImage	:	ITcVnImage;	(* Source image *)
		ipDestImage	:	REFERENCE TO ITcVnImage;	(* Destination image (Must be different from ipSrcImage! An appropriate destination image will be created if required.) *)
		nDiameter	:	DINT;	(* Diameter of the pixel neighborhood used for filtering (e.g. 5, 7, 9). If <= 0, it is automatically chosen dependend on fSigmaSpace. *)
		fSigmaColor	:	LREAL;	(* Sigma used for color space filtering (> 0). A larger value means that farther colors are mixed together. *)
		fSigmaSpace	:	LREAL;	(* Sigma used for coordinate space filtering (> 0). A larger value means that farther pixels can influence each other. *)
		hrPrev	:	HRESULT;	(* HRESULT indicating the result of previous operations (If SUCCEEDED(hrPrev) equals false, no operation is executed.) *)
	END_VAR

END_FUNCTION

// Functions/Image Filtering/F_VN_BilateralFilterExp

	{attribute 'TcIecLibraryType'}
	{attribute 'external_name' := 'F_VN_BilateralFilterExp_GUID_DD638786_5576_D234_70CF_F7DADAB6C09E'}
	(* Apply a Bilateral filter to smooth the image but preserve edges. (expert function) *)
	FUNCTION F_VN_BilateralFilterExp : HRESULT
	VAR_INPUT
		ipSrcImage	:	ITcVnImage;	(* Source image *)
		ipDestImage	:	REFERENCE TO ITcVnImage;	(* Destination image (Must be different from ipSrcImage! An appropriate destination image will be created if required.) *)
		nDiameter	:	DINT;	(* Diameter of the pixel neighborhood used for filtering (e.g. 5, 7, 9). If <= 0, it is automatically chosen dependend on fSigmaSpace. *)
		fSigmaColor	:	LREAL;	(* Sigma used for color space filtering (> 0). A larger value means that farther colors are mixed together. *)
		fSigmaSpace	:	LREAL;	(* Sigma used for coordinate space filtering (> 0). A larger value means that farther pixels can influence each other. *)
		eBorderType	:	ETcVnBorderInterpolationMethod;	(* Image border handling *)
		hrPrev	:	HRESULT;	(* HRESULT indicating the result of previous operations (If SUCCEEDED(hrPrev) equals false, no operation is executed.) *)
	END_VAR

END_FUNCTION

// Functions/Image Filtering/F_VN_BoxFilter

	{attribute 'TcIecLibraryType'}
	{attribute 'external_name' := 'F_VN_BoxFilter_GUID_E69755A6_8B2D_DF1E_4F41_0311CC50EAA8'}
	(* Apply a box filter to an image. *)
	FUNCTION F_VN_BoxFilter : HRESULT
	VAR_INPUT
		ipSrcImage	:	ITcVnImage;	(* Source image *)
		ipDestImage	:	REFERENCE TO ITcVnImage;	(* Destination image (An appropriate destination image will be created if required.) *)
		nFilterWidth	:	UDINT;	(* Filter width in pixels *)
		nFilterHeight	:	UDINT;	(* Filter height in pixels *)
		hrPrev	:	HRESULT;	(* HRESULT indicating the result of previous operations (If SUCCEEDED(hrPrev) equals false, no operation is executed.) *)
	END_VAR

END_FUNCTION

// Functions/Image Filtering/F_VN_BoxFilterExp

	{attribute 'TcIecLibraryType'}
	{attribute 'external_name' := 'F_VN_BoxFilterExp_GUID_BE35BE3C_685A_D86A_69F9_B319FFF2B795'}
	(* Apply a box filter to an image. (expert function) *)
	FUNCTION F_VN_BoxFilterExp : HRESULT
	VAR_INPUT
		ipSrcImage	:	ITcVnImage;	(* Source image *)
		ipDestImage	:	REFERENCE TO ITcVnImage;	(* Destination image (An appropriate destination image will be created if required.) *)
		nFilterWidth	:	UDINT;	(* Filter width in pixels *)
		nFilterHeight	:	UDINT;	(* Filter height in pixels *)
		eDestDepth	:	ETcVnElementType;	(* Destination image depth *)
	END_VAR
	VAR_IN_OUT
		aAnchor	:	TcVnPoint;	(* Anchor point of the kernel ([-1, -1] for center) *)
	END_VAR
	VAR_INPUT
		bNormalize	:	BOOL;	(* If true, the kernel is normalized by nFilterWidth * nFilterHeight *)
		eBorderType	:	ETcVnBorderInterpolationMethod;	(* Image border handling *)
		hrPrev	:	HRESULT;	(* HRESULT indicating the result of previous operations (If SUCCEEDED(hrPrev) equals false, no operation is executed.) *)
	END_VAR

END_FUNCTION

// Functions/Image Filtering/F_VN_BrightBorderObjects

	{attribute 'TcIecLibraryType'}
	{attribute 'external_name' := 'F_VN_BrightBorderObjects_GUID_C0BA5CAA_FDF5_D4FD_5590_697C119EFA93'}
	(* Find bright objects connected to the image border within a gray-scale single-channel image. *)
	FUNCTION F_VN_BrightBorderObjects : HRESULT
	VAR_INPUT
		ipSrcImage	:	ITcVnImage;	(* Source image (USINT, UINT, INT, REAL, or LREAL, 1 channel) *)
		ipDestImage	:	REFERENCE TO ITcVnImage;	(* Destination image (An appropriate destination image will be created if required.) *)
		hrPrev	:	HRESULT;	(* HRESULT indicating the result of previous operations (If SUCCEEDED(hrPrev) equals false, no operation is executed.) *)
	END_VAR

END_FUNCTION

// Functions/Image Filtering/F_VN_CreateStructuringElement

	{attribute 'TcIecLibraryType'}
	{attribute 'external_name' := 'F_VN_CreateStructuringElement_GUID_E2608966_D6B4_DF31_6D4F_8720564DC807'}
	(* Creates a structuring element for the usage with morphological operators and allocate an appropriate data buffer. The initial reference count is set to one if a new image interface is created and kept, otherwise. *)
	FUNCTION F_VN_CreateStructuringElement : HRESULT
	VAR_INPUT
		ipStructuringElement	:	REFERENCE TO ITcVnImage;	(* Returns the created structuring element (Non-zero interface pointers are reused.) *)
		eShape	:	ETcVnStructuringElementShape;	(* Shape of the structuring element (rectangle, cross, or ellipse) *)
		nWidth	:	UDINT;	(* Width *)
		nHeight	:	UDINT;	(* Height *)
		hrPrev	:	HRESULT;	(* HRESULT indicating the result of previous operations (If SUCCEEDED(hrPrev) equals false, no operation is executed.) *)
	END_VAR

END_FUNCTION

// Functions/Image Filtering/F_VN_CustomFilter

	{attribute 'TcIecLibraryType'}
	{attribute 'external_name' := 'F_VN_CustomFilter_GUID_062D9B85_A855_DF6A_4EBE_306A823F1C58'}
	(* Apply a custom filter to the image. *)
	FUNCTION F_VN_CustomFilter : HRESULT
	VAR_INPUT
		ipSrcImage	:	ITcVnImage;	(* Source image *)
		ipDestImage	:	REFERENCE TO ITcVnImage;	(* Destination image (An appropriate destination image will be created if required.) *)
		eDestDepth	:	ETcVnElementType;	(* Destination image depth *)
	END_VAR
	VAR_IN_OUT
		stKernel	:	TcVnMatrix;	(* Custom filter kernel with values of type REAL or LREAL *)
	END_VAR
	VAR_INPUT
		hrPrev	:	HRESULT;	(* HRESULT indicating the result of previous operations (If SUCCEEDED(hrPrev) equals false, no operation is executed.) *)
	END_VAR

END_FUNCTION

// Functions/Image Filtering/F_VN_CustomFilterExp

	{attribute 'TcIecLibraryType'}
	{attribute 'external_name' := 'F_VN_CustomFilterExp_GUID_2E3A926B_8F3F_DD0F_79EB_815DDCAF8ACA'}
	(* Apply a custom filter to the image. (expert function) *)
	FUNCTION F_VN_CustomFilterExp : HRESULT
	VAR_INPUT
		ipSrcImage	:	ITcVnImage;	(* Source image *)
		ipDestImage	:	REFERENCE TO ITcVnImage;	(* Destination image (An appropriate destination image will be created if required.) *)
		eDestDepth	:	ETcVnElementType;	(* Destination image depth *)
	END_VAR
	VAR_IN_OUT
		stKernel	:	TcVnMatrix;	(* Custom filter kernel with values of type REAL or LREAL *)
		aAnchor	:	TcVnPoint;	(* Anchor point of the kernel *)
	END_VAR
	VAR_INPUT
		fDelta	:	LREAL;	(* Value added to each pixel after filtering *)
		eBorderType	:	ETcVnBorderInterpolationMethod;	(* Image border handling *)
		hrPrev	:	HRESULT;	(* HRESULT indicating the result of previous operations (If SUCCEEDED(hrPrev) equals false, no operation is executed.) *)
	END_VAR

END_FUNCTION

// Functions/Image Filtering/F_VN_DarkBorderObjects

	{attribute 'TcIecLibraryType'}
	{attribute 'external_name' := 'F_VN_DarkBorderObjects_GUID_150638C3_24FF_D406_59DE_7207DF1FE4DD'}
	(* Find dark objects connected to the image border within a gray-scale single-channel image. (equivalent to filling holes) *)
	FUNCTION F_VN_DarkBorderObjects : HRESULT
	VAR_INPUT
		ipSrcImage	:	ITcVnImage;	(* Source image (USINT, UINT, INT, REAL, or LREAL, 1 channel) *)
		ipDestImage	:	REFERENCE TO ITcVnImage;	(* Destination image (An appropriate destination image will be created if required.) *)
		hrPrev	:	HRESULT;	(* HRESULT indicating the result of previous operations (If SUCCEEDED(hrPrev) equals false, no operation is executed.) *)
	END_VAR

END_FUNCTION

// Functions/Image Filtering/F_VN_FillHoles

	{attribute 'TcIecLibraryType'}
	{attribute 'external_name' := 'F_VN_FillHoles_GUID_70719E93_FD8E_D88B_6107_80117A24BEF3'}
	(* Fill holes within a gray-scale single-channel image. (equivalent to finding dark border objects) *)
	FUNCTION F_VN_FillHoles : HRESULT
	VAR_INPUT
		ipSrcImage	:	ITcVnImage;	(* Source image (USINT, UINT, INT, REAL, or LREAL, 1 channel) *)
		ipDestImage	:	REFERENCE TO ITcVnImage;	(* Destination image (An appropriate destination image will be created if required.) *)
		hrPrev	:	HRESULT;	(* HRESULT indicating the result of previous operations (If SUCCEEDED(hrPrev) equals false, no operation is executed.) *)
	END_VAR

END_FUNCTION

// Functions/Image Filtering/F_VN_GaussianFilter

	{attribute 'TcIecLibraryType'}
	{attribute 'external_name' := 'F_VN_GaussianFilter_GUID_A01527C3_D510_D586_4C2F_341A649AB36A'}
	(* Apply a Gaussian filter to smooth the image. *)
	FUNCTION F_VN_GaussianFilter : HRESULT
	VAR_INPUT
		ipSrcImage	:	ITcVnImage;	(* Source image *)
		ipDestImage	:	REFERENCE TO ITcVnImage;	(* Destination image (An appropriate destination image will be created if required.) *)
		nFilterWidth	:	UDINT;	(* Filter width in pixels (1, 3, 5, 7, ...) *)
		nFilterHeight	:	UDINT;	(* Filter height in pixels (1, 3, 5, 7, ...) *)
		hrPrev	:	HRESULT;	(* HRESULT indicating the result of previous operations (If SUCCEEDED(hrPrev) equals false, no operation is executed.) *)
	END_VAR

END_FUNCTION

// Functions/Image Filtering/F_VN_GaussianFilterExp

	{attribute 'TcIecLibraryType'}
	{attribute 'external_name' := 'F_VN_GaussianFilterExp_GUID_711C3136_A997_D1CF_4F62_43D5360D1994'}
	(* Apply a Gaussian filter to smooth the image. (expert function) *)
	FUNCTION F_VN_GaussianFilterExp : HRESULT
	VAR_INPUT
		ipSrcImage	:	ITcVnImage;	(* Source image *)
		ipDestImage	:	REFERENCE TO ITcVnImage;	(* Destination image (An appropriate destination image will be created if required.) *)
		nFilterWidth	:	UDINT;	(* Filter width in pixels (1, 3, 5, 7, ...) *)
		nFilterHeight	:	UDINT;	(* Filter height in pixels (1, 3, 5, 7, ...) *)
		fSigmaX	:	LREAL;	(* Gaussian kernel standard deviation in X direction (>= 0, automatically chosen if 0) *)
		fSigmaY	:	LREAL;	(* Gaussian kernel standard deviation in Y direction (>= 0, automatically chosen if 0) *)
		eBorderType	:	ETcVnBorderInterpolationMethod;	(* Image border handling *)
		hrPrev	:	HRESULT;	(* HRESULT indicating the result of previous operations (If SUCCEEDED(hrPrev) equals false, no operation is executed.) *)
	END_VAR

END_FUNCTION

// Functions/Image Filtering/F_VN_LaplacianFilter

	{attribute 'TcIecLibraryType'}
	{attribute 'external_name' := 'F_VN_LaplacianFilter_GUID_1744F7C5_9ECD_D130_77F7_FC0552AD20A9'}
	(* Apply a Laplacian filter to an image. *)
	FUNCTION F_VN_LaplacianFilter : HRESULT
	VAR_INPUT
		ipSrcImage	:	ITcVnImage;	(* Source image *)
		ipDestImage	:	REFERENCE TO ITcVnImage;	(* Destination image (An appropriate destination image will be created if required.) *)
		eDestDepth	:	ETcVnElementType;	(* Destination image depth *)
		hrPrev	:	HRESULT;	(* HRESULT indicating the result of previous operations (If SUCCEEDED(hrPrev) equals false, no operation is executed.) *)
	END_VAR

END_FUNCTION

// Functions/Image Filtering/F_VN_LaplacianFilterExp

	{attribute 'TcIecLibraryType'}
	{attribute 'external_name' := 'F_VN_LaplacianFilterExp_GUID_B5723878_DC26_D46C_70E1_70482EF49304'}
	(* Apply a Laplacian filter to an image. (expert function) *)
	FUNCTION F_VN_LaplacianFilterExp : HRESULT
	VAR_INPUT
		ipSrcImage	:	ITcVnImage;	(* Source image *)
		ipDestImage	:	REFERENCE TO ITcVnImage;	(* Destination image (An appropriate destination image will be created if required.) *)
		eDestDepth	:	ETcVnElementType;	(* Destination image depth *)
		nKernelSize	:	UDINT;	(* Aperture size used to compute the second-derivative filters (1, 3, 5, ..., 31) *)
		fScale	:	LREAL;	(* Scale factor for the computed derivative values *)
		fDelta	:	LREAL;	(* Delta value that is added to the results before storing them *)
		eBorderType	:	ETcVnBorderInterpolationMethod;	(* Image border handling *)
		hrPrev	:	HRESULT;	(* HRESULT indicating the result of previous operations (If SUCCEEDED(hrPrev) equals false, no operation is executed.) *)
	END_VAR

END_FUNCTION

// Functions/Image Filtering/F_VN_LocalMaxima

	{attribute 'TcIecLibraryType'}
	{attribute 'external_name' := 'F_VN_LocalMaxima_GUID_36CED361_9492_DC0E_4A0D_05A06FF2CB14'}
	(* Find local maxima in a gray-scale single-channel image. The found maxima are marked by a value of 1 in the destination image. *)
	FUNCTION F_VN_LocalMaxima : HRESULT
	VAR_INPUT
		ipSrcImage	:	ITcVnImage;	(* Source image (USINT or UINT, 1 channel) *)
		ipDestImage	:	REFERENCE TO ITcVnImage;	(* Destination image (Must be different from ipSrcImage! An appropriate destination image will be created if required.) *)
		hrPrev	:	HRESULT;	(* HRESULT indicating the result of previous operations (If SUCCEEDED(hrPrev) equals false, no operation is executed.) *)
	END_VAR

END_FUNCTION

// Functions/Image Filtering/F_VN_LocalMinima

	{attribute 'TcIecLibraryType'}
	{attribute 'external_name' := 'F_VN_LocalMinima_GUID_069EBDFC_0F10_D79E_5AC0_88B5BEB70BFB'}
	(* Find local minima in a gray-scale single-channel image. The found minima are marked by a value of 1 in the destination image. *)
	FUNCTION F_VN_LocalMinima : HRESULT
	VAR_INPUT
		ipSrcImage	:	ITcVnImage;	(* Source image (USINT or UINT, 1 channel) *)
		ipDestImage	:	REFERENCE TO ITcVnImage;	(* Destination image (Must be different from ipSrcImage! An appropriate destination image will be created if required.) *)
		hrPrev	:	HRESULT;	(* HRESULT indicating the result of previous operations (If SUCCEEDED(hrPrev) equals false, no operation is executed.) *)
	END_VAR

END_FUNCTION

// Functions/Image Filtering/F_VN_MedianFilter

	{attribute 'TcIecLibraryType'}
	{attribute 'external_name' := 'F_VN_MedianFilter_GUID_2D8DAC87_9773_DC7E_4167_1764713F62B3'}
	(* Apply a Median filter to an image. *)
	FUNCTION F_VN_MedianFilter : HRESULT
	VAR_INPUT
		ipSrcImage	:	ITcVnImage;	(* Source image (for nFilterSize 3 or 5: USINT, UINT, REAL. For bigger filters, only USINT is supported. *)
		ipDestImage	:	REFERENCE TO ITcVnImage;	(* Destination image (An appropriate destination image will be created if required.) *)
		nFilterSize	:	UDINT;	(* Size (width and height) of the filter (3, 5, 7, ...) *)
		hrPrev	:	HRESULT;	(* HRESULT indicating the result of previous operations (If SUCCEEDED(hrPrev) equals false, no operation is executed.) *)
	END_VAR

END_FUNCTION

// Functions/Image Filtering/F_VN_MorphologicalOperator

	{attribute 'TcIecLibraryType'}
	{attribute 'external_name' := 'F_VN_MorphologicalOperator_GUID_8786B0F7_F522_D1AC_6DEA_B623345CD034'}
	(* Apply a morphological operator. *)
	FUNCTION F_VN_MorphologicalOperator : HRESULT
	VAR_INPUT
		ipSrcImage	:	ITcVnImage;	(* Source image (only 1 channel supported for reconstruction operators) *)
		ipDestImage	:	REFERENCE TO ITcVnImage;	(* Destination image (An appropriate destination image will be created if required.) *)
		eOperator	:	ETcVnMorphologicalOperator;	(* Operator type *)
		ipStructuringElement	:	ITcVnImage;	(* Structuring element to be applied (Typically created via F_VN_CreateStructuringElement.) *)
		hrPrev	:	HRESULT;	(* HRESULT indicating the result of previous operations (If SUCCEEDED(hrPrev) equals false, no operation is executed.) *)
	END_VAR

END_FUNCTION

// Functions/Image Filtering/F_VN_RemoveLocalMaxima

	{attribute 'TcIecLibraryType'}
	{attribute 'external_name' := 'F_VN_RemoveLocalMaxima_GUID_56172991_A087_D4AB_6D55_446818348794'}
	(* Remove local maxima up to a given height from a gray-scale single-channel image. *)
	FUNCTION F_VN_RemoveLocalMaxima : HRESULT
	VAR_INPUT
		ipSrcImage	:	ITcVnImage;	(* Source image (USINT, UINT, INT, REAL, or LREAL, 1 channel) *)
		ipDestImage	:	REFERENCE TO ITcVnImage;	(* Destination image (An appropriate destination image will be created if required.) *)
		fHeight	:	LREAL;	(* Maximum height of the maxima to be removed (must be greater than 0) *)
		hrPrev	:	HRESULT;	(* HRESULT indicating the result of previous operations (If SUCCEEDED(hrPrev) equals false, no operation is executed.) *)
	END_VAR

END_FUNCTION

// Functions/Image Filtering/F_VN_RemoveLocalMinima

	{attribute 'TcIecLibraryType'}
	{attribute 'external_name' := 'F_VN_RemoveLocalMinima_GUID_E0B82E32_C5F7_DF23_58AB_A7FC386ED0F4'}
	(* Remove local minima up to a given height from a gray-scale single-channel image. *)
	FUNCTION F_VN_RemoveLocalMinima : HRESULT
	VAR_INPUT
		ipSrcImage	:	ITcVnImage;	(* Source image (USINT, UINT, INT, REAL, or LREAL, 1 channel) *)
		ipDestImage	:	REFERENCE TO ITcVnImage;	(* Destination image (An appropriate destination image will be created if required.) *)
		fHeight	:	LREAL;	(* Maximum height of the minima to be removed (must be greater than 0) *)
		hrPrev	:	HRESULT;	(* HRESULT indicating the result of previous operations (If SUCCEEDED(hrPrev) equals false, no operation is executed.) *)
	END_VAR

END_FUNCTION

// Functions/Image Filtering/F_VN_ScharrFilter

	{attribute 'TcIecLibraryType'}
	{attribute 'external_name' := 'F_VN_ScharrFilter_GUID_79F8CB90_B872_D9E4_43A8_908C130EBC68'}
	(* Calculates the first order derivative in x or y direction using a Scharr filter. *)
	FUNCTION F_VN_ScharrFilter : HRESULT
	VAR_INPUT
		ipSrcImage	:	ITcVnImage;	(* Source image *)
		ipDestImage	:	REFERENCE TO ITcVnImage;	(* Destination image (An appropriate destination image will be created if required.) *)
		eDestDepth	:	ETcVnElementType;	(* Destination image depth *)
		eFilterDirection	:	ETcVnFilterDirection;	(* Filter direction *)
		hrPrev	:	HRESULT;	(* HRESULT indicating the result of previous operations (If SUCCEEDED(hrPrev) equals false, no operation is executed.) *)
	END_VAR

END_FUNCTION

// Functions/Image Filtering/F_VN_ScharrFilterExp

	{attribute 'TcIecLibraryType'}
	{attribute 'external_name' := 'F_VN_ScharrFilterExp_GUID_51BA2996_DE04_D20D_47A3_88CD83463E40'}
	(* Calculates the first order derivative in x or y direction using a Scharr filter. (expert function) *)
	FUNCTION F_VN_ScharrFilterExp : HRESULT
	VAR_INPUT
		ipSrcImage	:	ITcVnImage;	(* Source image *)
		ipDestImage	:	REFERENCE TO ITcVnImage;	(* Destination image (An appropriate destination image will be created if required.) *)
		eDestDepth	:	ETcVnElementType;	(* Destination image depth *)
		eFilterDirection	:	ETcVnFilterDirection;	(* Filter direction *)
		fScale	:	LREAL;	(* Scale factor for the computed derivative values *)
		fDelta	:	LREAL;	(* Delta value that is added to the results prior to storing them in dest *)
		eBorderType	:	ETcVnBorderInterpolationMethod;	(* Image border handling *)
		hrPrev	:	HRESULT;	(* HRESULT indicating the result of previous operations (If SUCCEEDED(hrPrev) equals false, no operation is executed.) *)
	END_VAR

END_FUNCTION

// Functions/Image Filtering/F_VN_SeparableCustomFilter

	{attribute 'TcIecLibraryType'}
	{attribute 'external_name' := 'F_VN_SeparableCustomFilter_GUID_26A25BFD_C3D3_DB43_6161_872FEECDDE12'}
	(* Apply a separable custom filter to the image. *)
	FUNCTION F_VN_SeparableCustomFilter : HRESULT
	VAR_INPUT
		ipSrcImage	:	ITcVnImage;	(* Source image *)
		ipDestImage	:	REFERENCE TO ITcVnImage;	(* Destination image (An appropriate destination image will be created if required.) *)
		eDestDepth	:	ETcVnElementType;	(* Destination image depth *)
	END_VAR
	VAR_IN_OUT
		stKernelX	:	TcVnMatrix;	(* 1D custom row-filter kernel with values of type REAL or LREAL *)
		stKernelY	:	TcVnMatrix;	(* 1D custom column-filter kernel with values of type REAL or LREAL *)
	END_VAR
	VAR_INPUT
		hrPrev	:	HRESULT;	(* HRESULT indicating the result of previous operations (If SUCCEEDED(hrPrev) equals false, no operation is executed.) *)
	END_VAR

END_FUNCTION

// Functions/Image Filtering/F_VN_SeparableCustomFilterExp

	{attribute 'TcIecLibraryType'}
	{attribute 'external_name' := 'F_VN_SeparableCustomFilterExp_GUID_89767567_C202_D9D7_4A79_F3004FF852EC'}
	(* Apply a separable custom filter to the image. (expert function) *)
	FUNCTION F_VN_SeparableCustomFilterExp : HRESULT
	VAR_INPUT
		ipSrcImage	:	ITcVnImage;	(* Source image *)
		ipDestImage	:	REFERENCE TO ITcVnImage;	(* Destination image (An appropriate destination image will be created if required.) *)
		eDestDepth	:	ETcVnElementType;	(* Destination image depth *)
	END_VAR
	VAR_IN_OUT
		stKernelX	:	TcVnMatrix;	(* 1D custom row-filter kernel with values of type REAL or LREAL *)
		stKernelY	:	TcVnMatrix;	(* 1D custom column-filter kernel with values of type REAL or LREAL *)
		aAnchor	:	TcVnPoint;	(* Anchor point of the kernel *)
	END_VAR
	VAR_INPUT
		fDelta	:	LREAL;	(* Value added to each pixel after filtering *)
		eBorderType	:	ETcVnBorderInterpolationMethod;	(* Image border handling *)
		hrPrev	:	HRESULT;	(* HRESULT indicating the result of previous operations (If SUCCEEDED(hrPrev) equals false, no operation is executed.) *)
	END_VAR

END_FUNCTION

// Functions/Image Filtering/F_VN_SobelFilter

	{attribute 'TcIecLibraryType'}
	{attribute 'external_name' := 'F_VN_SobelFilter_GUID_3D9BE5A0_3C1A_D3F8_4354_64850ABA3B27'}
	(* Calculates the first, second, or mixed image derivatives using an extended Sobel filter. *)
	FUNCTION F_VN_SobelFilter : HRESULT
	VAR_INPUT
		ipSrcImage	:	ITcVnImage;	(* Source image *)
		ipDestImage	:	REFERENCE TO ITcVnImage;	(* Destination image (An appropriate destination image will be created if required.) *)
		eDestDepth	:	ETcVnElementType;	(* Destination image depth *)
		nXOrder	:	UDINT;	(* Order of the x-derivative (0, 1, 2) *)
		nYOrder	:	UDINT;	(* Order of the y-derivative (0, 1, 2) *)
		hrPrev	:	HRESULT;	(* HRESULT indicating the result of previous operations (If SUCCEEDED(hrPrev) equals false, no operation is executed.) *)
	END_VAR

END_FUNCTION

// Functions/Image Filtering/F_VN_SobelFilterExp

	{attribute 'TcIecLibraryType'}
	{attribute 'external_name' := 'F_VN_SobelFilterExp_GUID_BEF3CEFC_5763_DE67_684A_5322EB10B590'}
	(* Calculates the first, second, third, or mixed image derivatives using an extended Sobel filter. (expert function) *)
	FUNCTION F_VN_SobelFilterExp : HRESULT
	VAR_INPUT
		ipSrcImage	:	ITcVnImage;	(* Source image *)
		ipDestImage	:	REFERENCE TO ITcVnImage;	(* Destination image (An appropriate destination image will be created if required.) *)
		eDestDepth	:	ETcVnElementType;	(* Destination image depth *)
		nXOrder	:	UDINT;	(* Order of the x-derivative (must be < nKernelSize) *)
		nYOrder	:	UDINT;	(* Order of the y-derivative (must be < nKernelSize) *)
		nKernelSize	:	UDINT;	(* Size of the extended Sobel kernel (3, 5, 7, ..., 31) *)
		fScale	:	LREAL;	(* Scale factor for the computed derivative values *)
		fDelta	:	LREAL;	(* Delta value that is added to the results prior to storing them in dest *)
		eBorderType	:	ETcVnBorderInterpolationMethod;	(* Image border handling *)
		hrPrev	:	HRESULT;	(* HRESULT indicating the result of previous operations (If SUCCEEDED(hrPrev) equals false, no operation is executed.) *)
	END_VAR

END_FUNCTION

// Functions/Image Filtering/F_VN_VarianceFilter

	{attribute 'TcIecLibraryType'}
	{attribute 'external_name' := 'F_VN_VarianceFilter_GUID_3771ACE7_A83B_D4DE_50D9_35056A07A35C'}
	(* Calculates the local variance of an image. *)
	FUNCTION F_VN_VarianceFilter : HRESULT
	VAR_INPUT
		ipSrcImage	:	ITcVnImage;	(* Source image. Only TCVN_ET_USINT Type is supported.  *)
		ipDestImage	:	REFERENCE TO ITcVnImage;	(* Destination image of type TCVN_ET_UINT (An appropriate destination image will be created if required.) *)
		nKernelSize	:	UDINT;	(* Size of the kernel *)
		hrPrev	:	HRESULT;	(* HRESULT indicating the result of previous operations (If SUCCEEDED(hrPrev) equals false, no operation is executed.) *)
	END_VAR

END_FUNCTION

// Functions/Image Filtering/F_VN_VarianceFilterExp

	{attribute 'TcIecLibraryType'}
	{attribute 'external_name' := 'F_VN_VarianceFilterExp_GUID_7D79AC61_7A78_DCFB_7472_C1E2F20752E3'}
	(* Calculates the local variance of an image. (expert function) *)
	FUNCTION F_VN_VarianceFilterExp : HRESULT
	VAR_INPUT
		ipSrcImage	:	ITcVnImage;	(* Source image. Only TCVN_ET_USINT Type is supported. *)
		ipDestImage	:	REFERENCE TO ITcVnImage;	(* Destination image of type TCVN_ET_UINT (An appropriate destination image will be created if required.) *)
		nKernelSize	:	UDINT;	(* Size of the kernel *)
		fScale	:	LREAL;	(* Scale factor for the computed variance values *)
		eBorderType	:	ETcVnBorderInterpolationMethod;	(* Image border handling *)
		hrPrev	:	HRESULT;	(* HRESULT indicating the result of previous operations (If SUCCEEDED(hrPrev) equals false, no operation is executed.) *)
	END_VAR

END_FUNCTION

// Functions/Miscellaneous/F_VN_CheckFunctionInitialization

	{attribute 'TcIecLibraryType'}
	{attribute 'external_name' := 'F_VN_CheckFunctionInitialization_GUID_1930A7E8_61B1_DE6C_56D4_87D5B4B2C546'}
	(* Check if a function is initialized with the specified options. *)
	FUNCTION F_VN_CheckFunctionInitialization : HRESULT
	VAR_INPUT
		eFunction	:	ETcVnInitializableFunction;	(* Initializable function *)
		nOptions	:	ULINT;	(* Initialization options for the function *)
		hrPrev	:	HRESULT;	(* HRESULT indicating the result of previous operations (If SUCCEEDED(hrPrev) equals false, no operation is executed.) *)
	END_VAR

END_FUNCTION

// Functions/Miscellaneous/F_VN_ClipLineToBoundary

